// TIA Portal project "DigitalTwin_Selecao_de_Pecas" (V14)
// Trabalho de conclusão de curso, um gêmeo digital de um processo de seleção de peças em uma transportadora

(* hardware
DEVICE "S7-1200 station_3"  S7-1200 Station
   slot 0: "Rack_0"  S7-1200 Rack  Rack  V1.0
   slot 1: "S71200 Físico"  CPU 1214C DC/DC/DC  6ES7 214-1AG40-0XB0  V4.2
   slot 3: "AQ 1x12BIT_1"  AQ1 signal board  6ES7 232-4HA30-0XB0  V1.0
DEVICE "S71500/ET200MP station_2"  S7-1500 station
   slot 0: "Rail_0"  Rack  6ES7 590-1***0-0AA0
   slot 1: "PLCSim Adavanced"  CPU 1511-1 PN  6ES7 511-1AK01-0AB0  V2.1
      slot 3: "CPU display_1"  6ES7591-1AA00-0AA0
*)

// ===== PLC "S71200 Físico"  CPU 1214C DC/DC/DC =====

VAR_GLOBAL   // PLC tag table "Default tag table"
   "System_Byte" AT %MB1 : Byte;
   "FirstScan" AT %M1.0 : Bool;
   "DiagStatusUpdate" AT %M1.1 : Bool;
   "AlwaysTRUE" AT %M1.2 : Bool;
   "AlwaysFALSE" AT %M1.3 : Bool;
   "System_Byte(1)" AT %MB1 : Byte;
   "Clock_Byte" AT %MB0 : Byte;
   "Clock_10Hz" AT %M0.0 : Bool;
   "Clock_5Hz" AT %M0.1 : Bool;
   "Clock_2.5Hz" AT %M0.2 : Bool;
   "Clock_2Hz" AT %M0.3 : Bool;
   "Clock_1.25Hz" AT %M0.4 : Bool;
   "Clock_1Hz" AT %M0.5 : Bool;
   "Clock_0.625Hz" AT %M0.6 : Bool;
   "Clock_0.5Hz" AT %M0.7 : Bool;
END_VAR

VAR_GLOBAL   // PLC tag table "Entradas Digitais"
   "DIn_ATD001_PrsMat01" AT %I0.0 : Bool;   // Esteira transportadora (ET-111) - Presença de material (tamanho maior)
   "DIn_ATD001_PrsMat02" AT %I0.1 : Bool;   // Esteira transportadora (ET-111) - Presença de material (tamanho médio)
   "DIn_ATD001_PrsMat03" AT %I0.2 : Bool;   // Esteira transportadora (ET-111) - Presença de material (tamanho menor)
   "DIn_ATD001_PrsMat04" AT %I0.3 : Bool;   // Esteira transportadora (ET-111) - Presença de material (Capacitivo)
   "DIn_ATD001_PrsMat05" AT %I0.4 : Bool;   // Esteira transportadora (ET-111) - Presença de material (Indutivo)
   "DIn_ATD001_PrsMat06" AT %I0.5 : Bool;   // Esteira transportadora (ET-111) - Presença de material (Setor A)
   "DIn_ATD001_PrsMat07" AT %I0.6 : Bool;   // Esteira transportadora (ET-111) - Presença de material (Setor B)
   "DIn_ATD001_PrsMat08" AT %I0.7 : Bool;   // Esteira transportadora (ET-111) - Presença de material (Setor C)
   "DIn_ATD001_PrsMat09" AT %I1.0 : Bool;   // Esteira transportadora (ET-111) - Presença de material (Setor D)
   "Din_Geral_AtvEmg" AT %I1.1 : Bool;   // Geral - Ativa condição de emergência [NF]
   "Din_Geral_AtvRst" AT %I1.2 : Bool;   // Geral - Ativa reset
END_VAR

VAR_GLOBAL   // PLC tag table "Saídas Analógicas"
   "Dou_ATD001_LigElm" AT %QW64 : UInt;   // Esteira transportadora (ET-111) - Liga elemento (Esteira A)
END_VAR

VAR_GLOBAL   // PLC tag table "Saídas Digitais"
   "Dou_ATD002_AvnElm" AT %Q0.0 : Bool;   // Pistão Separador A (PI-111) - Avança elemento
   "Dou_ATD003_AvnElm" AT %Q0.1 : Bool;   // Pistão Separador B (PI-112) - Avança elemento
   "Dou_ATD004_AvnElm" AT %Q0.2 : Bool;   // Pistão Separador C (PI-113) - Avança elemento
   "Dou_ATD004_RcuElm" AT %Q0.3 : Bool;   // Pistão Separador C (PI-113) - Recua elemento
END_VAR

// folder: System blocks/Program resources

DATA_BLOCK "EES001_DlyDsv01"   // DB4
{ S7_Optimized_Access := 'TRUE' }
AUTHOR : Simatic
FAMILY : IEC
NAME : IEC_TMR
VERSION : 1.0
// stored: InstanceOfName IEC_TIMER
"IEC_TIMER"
BEGIN
END_DATA_BLOCK

// folder: VARIÁVEIS/0 - Gerais

DATA_BLOCK "EDG"   // DB1
TITLE = Detecção de Bordas
{ S7_Optimized_Access := 'TRUE' }
VERSION : 0.1
   VAR
      GRP001_DtcPos01 : Bool;   // Geral - Detecção positiva
      EES001_DtcPos01 : Bool;   // Selecionador de Peças - Detecção positiva
      EES001_DtcPos02 : Bool;   // Selecionador de Peças - Detecção positiva (Aux)
      EES001_DtcPos03 : Bool;   // Selecionador de Peças - Detecção positiva (Tempo de transporte)
   END_VAR
BEGIN
END_DATA_BLOCK

DATA_BLOCK "TMR"   // DB2
TITLE = Temporizadores
{ S7_Optimized_Access := 'TRUE' }
VERSION : 0.1
   VAR
      EES001_DlyAtv01 : IEC_TIMER;   // Selecionador de Peças - Atraso para ativar
      EES001_DlyAtv02 : IEC_TIMER;   // Selecionador de Peças - Atraso para ativar
      EES001_DlyAtv03 : IEC_TIMER;   // Selecionador de Peças - Atraso para ativar
      ATD003_DlyAtv01 : IEC_TIMER;   // Pistão Separador B - Atraso para ativar
      EES001_DlyDsv01 : IEC_TIMER;   // Selecionador de Peças - Atraso para desativar
      EES001_DlyDsv02 : IEC_TIMER;   // Selecionador de Peças - Atraso para desativar (Recuar Pistão C)
      ATD004_DlyAtv01 : IEC_TIMER;   // Pistão Separador C - Atraso para ativar (Avançar)
      EES001_DlyAtv04 : IEC_TIMER;   // Selecionador de Peças - Atraso para ativar (Tempo de transporte)
   END_VAR
BEGIN
END_DATA_BLOCK

DATA_BLOCK "CTR"   // DB3
TITLE = Contadores
{ S7_Optimized_Access := 'TRUE' }
VERSION : 0.1
   VAR
      EES001_CntUnd01 : IEC_UCOUNTER;   // Selecionador de Peças - Conta unidades (Setor A)
      EES001_CntUnd02 : IEC_UCOUNTER;   // Selecionador de Peças - Conta unidades (Setor B)
      EES001_CntUnd03 : IEC_UCOUNTER;   // Selecionador de Peças - Conta unidades (Setor C)
      EES001_CntUnd04 : IEC_UCOUNTER;   // Selecionador de Peças - Conta unidades (Setor D)
   END_VAR
BEGIN
END_DATA_BLOCK

// folder: VARIÁVEIS/1 - Comandos

DATA_BLOCK "CmdEsp"   // DB110
{ S7_Optimized_Access := 'FALSE' }
VERSION : 0.1
BEGIN
END_DATA_BLOCK

DATA_BLOCK "CmdGrp"   // DB120
{ S7_Optimized_Access := 'FALSE' }
VERSION : 0.1
   VAR
      GRP001 : Struct   // Geral
         RrmElm : Bool := false;   // Geral - Rearma Elemento
         SelAut : Bool := false;   // Geral - Seleciona modo automático para todos atuadores
         SelMaa : Bool := false;   // Geral - Seleciona modo manual para todos atuadores
         xd0r3 : Bool := false;   // Reserva
         xd0r4 : Bool := false;   // Reserva
         xd0r5 : Bool := false;   // Reserva
         xd0r6 : Bool := false;   // Reserva
         xd0r7 : Bool := false;   // Reserva
         xd1r0 : Bool := false;   // Reserva
         xd1r1 : Bool := false;   // Reserva
         xd1r2 : Bool := false;   // Reserva
         xd1r3 : Bool := false;   // Reserva
         xd1r4 : Bool := false;   // Reserva
         xd1r5 : Bool := false;   // Reserva
         xd1r6 : Bool := false;   // Reserva
         xd1r7 : Bool := false;   // Reserva
      END_STRUCT;
   END_VAR
BEGIN
END_DATA_BLOCK

DATA_BLOCK "CmdAtd"   // DB130
TITLE = Comandos
{ S7_Optimized_Access := 'FALSE' }
VERSION : 0.1
   VAR
      ATD001 : Struct   // Esteira Transportadora (ET-111)
         SelAut : Bool;   // Esteira Transportadora (ET-111) - Seleciona modo automático
         SelMaa : Bool := false;   // Esteira Transportadora (ET-111) - Seleciona modo manual
         LigElm : Bool := false;   // Esteira Transportadora (ET-111) - Liga elemento
         DsgElm : Bool := false;   // Esteira Transportadora (ET-111) - Desliga elemento
         xd0r4 : Bool := false;   // Reserva
         xd0r5 : Bool := false;   // Reserva
         xd0r6 : Bool := false;   // Reserva
         xd0r7 : Bool := false;   // Reserva
         xd1r0 : Bool;   // Reserva
         xd1r1 : Bool := false;   // Reserva
         xd1r2 : Bool := false;   // Reserva
         xd1r3 : Bool := false;   // Reserva
         xd1r4 : Bool := false;   // Reserva
         xd1r5 : Bool := false;   // Reserva
         xd1r6 : Bool := false;   // Reserva
         xd1r7 : Bool := false;   // Reserva
      END_STRUCT;
      ATD002 : Struct   // Pistão Separador A (PI-111)
         SelAut : Bool := false;   // Pistão Separador A (PI-111) - Seleciona modo automático
         SelMaa : Bool := false;   // Pistão Separador A (PI-111) - Seleciona modo manual
         AvnElm : Bool := false;   // Pistão Separador A (PI-111) - Avança elemento
         RcuElm : Bool := false;   // Pistão Separador A (PI-111) - Recua elemento
         xd0r4 : Bool := false;   // Reserva
         xd0r5 : Bool := false;   // Reserva
         xd0r6 : Bool := false;   // Reserva
         xd0r7 : Bool := false;   // Reserva
         xd1r0 : Bool := false;   // Reserva
         xd1r1 : Bool := false;   // Reserva
         xd1r2 : Bool := false;   // Reserva
         xd1r3 : Bool := false;   // Reserva
         xd1r4 : Bool := false;   // Reserva
         xd1r5 : Bool := false;   // Reserva
         xd1r6 : Bool := false;   // Reserva
         xd1r7 : Bool := false;   // Reserva
      END_STRUCT;
      ATD003 : Struct   // Pistão Separador B (PI-112)
         SelAut : Bool := false;   // Pistão Separador B (PI-112) - Seleciona modo automático
         SelMaa : Bool := false;   // Pistão Separador B (PI-112) - Seleciona modo manual
         AvnElm : Bool := false;   // Pistão Separador B (PI-112) - Avança elemento
         RcuElm : Bool := false;   // Pistão Separador B (PI-112) - Recua elemento
         xd0r4 : Bool := false;   // Reserva
         xd0r5 : Bool := false;   // Reserva
         xd0r6 : Bool := false;   // Reserva
         xd0r7 : Bool := false;   // Reserva
         xd1r0 : Bool := false;   // Reserva
         xd1r1 : Bool := false;   // Reserva
         xd1r2 : Bool := false;   // Reserva
         xd1r3 : Bool := false;   // Reserva
         xd1r4 : Bool := false;   // Reserva
         xd1r5 : Bool := false;   // Reserva
         xd1r6 : Bool := false;   // Reserva
         xd1r7 : Bool := false;   // Reserva
      END_STRUCT;
      ATD004 : Struct   // Pistão Separador C (PI-113)
         SelAut : Bool := false;   // Pistão Separador C (PI-113) - Seleciona modo automático
         SelMaa : Bool := false;   // Pistão Separador C (PI-113) - Seleciona modo manual
         AvnElm : Bool := false;   // Pistão Separador C (PI-113) - Avança elemento
         RcuElm : Bool := false;   // Pistão Separador C (PI-113) - Recua elemento
         xd0r4 : Bool := false;   // Reserva
         xd0r5 : Bool := false;   // Reserva
         xd0r6 : Bool := false;   // Reserva
         xd0r7 : Bool := false;   // Reserva
         xd1r0 : Bool := false;   // Reserva
         xd1r1 : Bool := false;   // Reserva
         xd1r2 : Bool := false;   // Reserva
         xd1r3 : Bool := false;   // Reserva
         xd1r4 : Bool := false;   // Reserva
         xd1r5 : Bool := false;   // Reserva
         xd1r6 : Bool := false;   // Reserva
         xd1r7 : Bool := false;   // Reserva
      END_STRUCT;
   END_VAR
BEGIN
END_DATA_BLOCK

DATA_BLOCK "CmdEes"   // DB160
{ S7_Optimized_Access := 'FALSE' }
VERSION : 0.1
   VAR
      EES001 : Struct   // Selecionador de Peças
         RrmElm : Bool := false;   // Selecionador de Peças - Rearma Elmento
         RmvPcs01 : Bool := false;   // Selecionador de Peças - Remove Peças (Setor A)
         RmvPcs02 : Bool := false;   // Selecionador de Peças - Remove Peças (Setor B)
         RmvPcs03 : Bool := false;   // Selecionador de Peças - Remove Peças (Setor C)
         RmvPcs04 : Bool := false;   // Selecionador de Peças - Remove Peças (Setor D)
         RstPcs : Bool := false;   // Selecionador de Peças - Reseta quantidade de Peças
         xd0r6 : Bool := false;   // Reserva
         xd0r7 : Bool := false;   // Reserva
         xd1r0 : Bool := false;   // Reserva
         xd1r1 : Bool := false;   // Reserva
         xd1r2 : Bool := false;   // Reserva
         xd1r3 : Bool := false;   // Reserva
         xd1r4 : Bool := false;   // Reserva
         xd1r5 : Bool := false;   // Reserva
         xd1r6 : Bool := false;   // Reserva
         xd1r7 : Bool := false;   // Reserva
      END_STRUCT;
   END_VAR
BEGIN
END_DATA_BLOCK

// folder: VARIÁVEIS/2 - Estados

DATA_BLOCK "SttEsp"   // DB210
{ S7_Optimized_Access := 'FALSE' }
VERSION : 0.1
BEGIN
END_DATA_BLOCK

DATA_BLOCK "SttGrp"   // DB220
{ S7_Optimized_Access := 'FALSE' }
VERSION : 0.1
   VAR
      GRP001 : Struct   // Geral
         xd0r0 : Bool := false;   // Reserva
         xd0r1 : Bool := false;   // Reserva
         xd0r2 : Bool := false;   // Reserva
         xd0r3 : Bool := false;   // Reserva
         xd0r4 : Bool := false;   // Reserva
         xd0r5 : Bool := false;   // Reserva
         xd0r6 : Bool := false;   // Reserva
         xd0r7 : Bool := false;   // Reserva
         xd1r0 : Bool := false;   // Reserva
         xd1r1 : Bool := false;   // Reserva
         xd1r2 : Bool := false;   // Reserva
         xd1r3 : Bool := false;   // Reserva
         xd1r4 : Bool := false;   // Reserva
         xd1r5 : Bool := false;   // Reserva
         xd1r6 : Bool := false;   // Reserva
         xd1r7 : Bool := false;   // Reserva
      END_STRUCT;
   END_VAR
BEGIN
END_DATA_BLOCK

DATA_BLOCK "SttAtd"   // DB230
TITLE = Estados de Atuadores
{ S7_Optimized_Access := 'FALSE' }
VERSION : 0.1
   VAR
      ATD001 : Struct   // Esteira Transportadora (ET-111)
         AutSel : Bool := false;   // Esteira Transportadora (ET-111) - Modo automático selecionado
         MaaSel : Bool := false;   // Esteira Transportadora (ET-111) - Modo manual selecionado
         ElmLig : Bool := false;   // Esteira Transportadora (ET-111) - Elemento ligado
         BlqLig : Bool := false;   // Esteira Transportadora (ET-111) - Bloqueado para ligar
         xd0r4 : Bool := false;   // Reserva
         xd0r5 : Bool := false;   // Reserva
         xd0r6 : Bool := false;   // Reserva
         xd0r7 : Bool := false;   // Reserva
         xd1r0 : Bool := false;   // Reserva
         xd1r1 : Bool := false;   // Reserva
         xd1r2 : Bool := false;   // Reserva
         xd1r3 : Bool := false;   // Reserva
         xd1r4 : Bool := false;   // Reserva
         xd1r5 : Bool := false;   // Reserva
         xd1r6 : Bool := false;   // Reserva
         xd1r7 : Bool := false;   // Reserva
      END_STRUCT;
      ATD002 : Struct   // Pistão Separador A (PI-111)
         AutSel : Bool := false;   // Pistão Separador A (PI-111) - Modo automático selecionado
         MaaSel : Bool := false;   // Pistão Separador A (PI-111) - Modo manual selecionado
         PosAvn : Bool := false;   // Pistão Separador A (PI-111) - Elemento avançado
         BlqAvn : Bool := false;   // Pistão Separador A (PI-111) - Bloqueado para avançar
         xd0r4 : Bool := false;   // Reserva
         xd0r5 : Bool := false;   // Reserva
         xd0r6 : Bool := false;   // Reserva
         xd0r7 : Bool := false;   // Reserva
         xd1r0 : Bool := false;   // Reserva
         xd1r1 : Bool := false;   // Reserva
         xd1r2 : Bool := false;   // Reserva
         xd1r3 : Bool := false;   // Reserva
         xd1r4 : Bool := false;   // Reserva
         xd1r5 : Bool := false;   // Reserva
         xd1r6 : Bool := false;   // Reserva
         xd1r7 : Bool := false;   // Reserva
      END_STRUCT;
      ATD003 : Struct   // Pistão Separador B (PI-112)
         AutSel : Bool := false;   // Pistão Separador B (PI-112) - Modo automático selecionado
         MaaSel : Bool := false;   // Pistão Separador B (PI-112) - Modo manual selecionado
         PosAvn : Bool := false;   // Pistão Separador B (PI-112) - Elemento avançado
         BlqAvn : Bool := false;   // Pistão Separador B (PI-112) - Bloqueado para Bloqueado para avançar
         xd0r4 : Bool := false;   // Reserva
         xd0r5 : Bool := false;   // Reserva
         xd0r6 : Bool := false;   // Reserva
         xd0r7 : Bool := false;   // Reserva
         xd1r0 : Bool := false;   // Reserva
         xd1r1 : Bool := false;   // Reserva
         xd1r2 : Bool := false;   // Reserva
         xd1r3 : Bool := false;   // Reserva
         xd1r4 : Bool := false;   // Reserva
         xd1r5 : Bool := false;   // Reserva
         xd1r6 : Bool := false;   // Reserva
         xd1r7 : Bool := false;   // Reserva
      END_STRUCT;
      ATD004 : Struct   // Pistão Separador C (PI-113)
         AutSel : Bool := false;   // Pistão Separador C (PI-113) - Modo automático selecionado
         MaaSel : Bool := false;   // Pistão Separador C (PI-113) - Modo manual selecionado
         PosAvn : Bool := false;   // Pistão Separador C (PI-113) - Elemento avançado
         BlqAvn : Bool := false;   // Pistão Separador C (PI-113) - Bloqueado para avançar
         PosRcu : Bool := false;   // Pistão Separador C (PI-113) - Elemento recuado
         BlqRcu : Bool := false;   // Pistão Separador C (PI-113) - Bloqueado para recuar
         xd0r6 : Bool := false;   // Reserva
         xd0r7 : Bool := false;   // Reserva
         xd1r0 : Bool := false;   // Reserva
         xd1r1 : Bool := false;   // Reserva
         xd1r2 : Bool := false;   // Reserva
         xd1r3 : Bool := false;   // Reserva
         xd1r4 : Bool := false;   // Reserva
         xd1r5 : Bool := false;   // Reserva
         xd1r6 : Bool := false;   // Reserva
         xd1r7 : Bool := false;   // Reserva
      END_STRUCT;
   END_VAR
BEGIN
END_DATA_BLOCK

DATA_BLOCK "SttEes"   // DB260
{ S7_Optimized_Access := 'FALSE' }
VERSION : 0.1
   VAR
      EES001 : Struct   // Selecionador de Peças
         ElmDef : Bool := false;   // Selecionador de Peças - Elmento com Defeito
         xd0r1 : Bool := false;   // Reserva
         xd0r2 : Bool := false;   // Reserva
         xd0r3 : Bool := false;   // Reserva
         xd0r4 : Bool := false;   // Reserva
         xd0r5 : Bool := false;   // Reserva
         xd0r6 : Bool := false;   // Reserva
         xd0r7 : Bool := false;   // Reserva
         xd1r0 : Bool := false;   // Reserva
         xd1r1 : Bool := false;   // Reserva
         xd1r2 : Bool := false;   // Reserva
         xd1r3 : Bool := false;   // Reserva
         xd1r4 : Bool := false;   // Reserva
         xd1r5 : Bool := false;   // Reserva
         xd1r6 : Bool := false;   // Reserva
         xd1r7 : Bool := false;   // Reserva
      END_STRUCT;
   END_VAR
BEGIN
END_DATA_BLOCK

// folder: VARIÁVEIS/3 - Alarmes

DATA_BLOCK "AlrEsp"   // DB310
{ S7_Optimized_Access := 'FALSE' }
VERSION : 0.1
BEGIN
END_DATA_BLOCK

DATA_BLOCK "AlrGrp"   // DB320
{ S7_Optimized_Access := 'FALSE' }
VERSION : 0.1
   VAR
      GRP001 : Struct   // Geral
         EmgAtv : Bool := false;   // Geral - Condição de Emergência Ativada
         xd0r1 : Bool := false;   // Reserva
         xd0r2 : Bool := false;   // Reserva
         xd0r3 : Bool := false;   // Reserva
         xd0r4 : Bool := false;   // Reserva
         xd0r5 : Bool := false;   // Reserva
         xd0r6 : Bool := false;   // Reserva
         xd0r7 : Bool := false;   // Reserva
         xd1r0 : Bool := false;   // Reserva
         xd1r1 : Bool := false;   // Reserva
         xd1r2 : Bool := false;   // Reserva
         xd1r3 : Bool := false;   // Reserva
         xd1r4 : Bool := false;   // Reserva
         xd1r5 : Bool := false;   // Reserva
         xd1r6 : Bool := false;   // Reserva
         xd1r7 : Bool := false;   // Reserva
      END_STRUCT;
   END_VAR
BEGIN
END_DATA_BLOCK

DATA_BLOCK "AlrAtd"   // DB330
TITLE = Alarmes de Atuadores
{ S7_Optimized_Access := 'FALSE' }
VERSION : 0.1
   VAR
      ATD001 : Struct   // Esteira Transportadora (ET-111)
         xd0r0 : Bool := false;   // Reserva
         xd0r1 : Bool := false;   // Reserva
         xd0r2 : Bool := false;   // Reserva
         xd0r3 : Bool := false;   // Reserva
         xd0r4 : Bool := false;   // Reserva
         xd0r5 : Bool := false;   // Reserva
         xd0r6 : Bool := false;   // Reserva
         xd0r7 : Bool := false;   // Reserva
         xd1r0 : Bool := false;   // Reserva
         xd1r1 : Bool := false;   // Reserva
         xd1r2 : Bool := false;   // Reserva
         xd1r3 : Bool := false;   // Reserva
         xd1r4 : Bool := false;   // Reserva
         xd1r5 : Bool := false;   // Reserva
         xd1r6 : Bool := false;   // Reserva
         xd1r7 : Bool := false;   // Reserva
      END_STRUCT;
      ATD002 : Struct   // Pistão Separador A (PI-111)
         xd0r0 : Bool := false;   // Reserva
         xd0r1 : Bool := false;   // Reserva
         xd0r2 : Bool := false;   // Reserva
         xd0r3 : Bool := false;   // Reserva
         xd0r4 : Bool := false;   // Reserva
         xd0r5 : Bool := false;   // Reserva
         xd0r6 : Bool := false;   // Reserva
         xd0r7 : Bool := false;   // Reserva
         xd1r0 : Bool := false;   // Reserva
         xd1r1 : Bool := false;   // Reserva
         xd1r2 : Bool := false;   // Reserva
         xd1r3 : Bool := false;   // Reserva
         xd1r4 : Bool := false;   // Reserva
         xd1r5 : Bool := false;   // Reserva
         xd1r6 : Bool := false;   // Reserva
         xd1r7 : Bool := false;   // Reserva
      END_STRUCT;
      ATD003 : Struct   // Pistão Separador B (PI-112)
         xd0r0 : Bool := false;   // Reserva
         xd0r1 : Bool := false;   // Reserva
         xd0r2 : Bool := false;   // Reserva
         xd0r3 : Bool := false;   // Reserva
         xd0r4 : Bool := false;   // Reserva
         xd0r5 : Bool := false;   // Reserva
         xd0r6 : Bool := false;   // Reserva
         xd0r7 : Bool := false;   // Reserva
         xd1r0 : Bool := false;   // Reserva
         xd1r1 : Bool := false;   // Reserva
         xd1r2 : Bool := false;   // Reserva
         xd1r3 : Bool := false;   // Reserva
         xd1r4 : Bool := false;   // Reserva
         xd1r5 : Bool := false;   // Reserva
         xd1r6 : Bool := false;   // Reserva
         xd1r7 : Bool := false;   // Reserva
      END_STRUCT;
      ATD004 : Struct   // Pistão Separador C (PI-113)
         xd0r0 : Bool := false;   // Reserva
         xd0r1 : Bool := false;   // Reserva
         xd0r2 : Bool := false;   // Reserva
         xd0r3 : Bool := false;   // Reserva
         xd0r4 : Bool := false;   // Reserva
         xd0r5 : Bool := false;   // Reserva
         xd0r6 : Bool := false;   // Reserva
         xd0r7 : Bool := false;   // Reserva
         xd1r0 : Bool := false;   // Reserva
         xd1r1 : Bool := false;   // Reserva
         xd1r2 : Bool := false;   // Reserva
         xd1r3 : Bool := false;   // Reserva
         xd1r4 : Bool := false;   // Reserva
         xd1r5 : Bool := false;   // Reserva
         xd1r6 : Bool := false;   // Reserva
         xd1r7 : Bool := false;   // Reserva
      END_STRUCT;
   END_VAR
BEGIN
END_DATA_BLOCK

DATA_BLOCK "AlrEes"   // DB360
{ S7_Optimized_Access := 'FALSE' }
VERSION : 0.1
   VAR
      EES001 : Struct   // Selecionador de Peças
         LimExc : Bool := false;   // Selecionador de Peças - Limite Excedido (Mais de uma peça em transporte)
         xd0r1 : Bool := false;   // Reserva
         xd0r2 : Bool := false;   // Reserva
         xd0r3 : Bool := false;   // Reserva
         xd0r4 : Bool := false;   // Reserva
         xd0r5 : Bool := false;   // Reserva
         xd0r6 : Bool := false;   // Reserva
         xd0r7 : Bool := false;   // Reserva
         xd1r0 : Bool := false;   // Reserva
         xd1r1 : Bool := false;   // Reserva
         xd1r2 : Bool := false;   // Reserva
         xd1r3 : Bool := false;   // Reserva
         xd1r4 : Bool := false;   // Reserva
         xd1r5 : Bool := false;   // Reserva
         xd1r6 : Bool := false;   // Reserva
         xd1r7 : Bool := false;   // Reserva
      END_STRUCT;
   END_VAR
BEGIN
END_DATA_BLOCK

// folder: VARIÁVEIS/4 - Intertravamentos

DATA_BLOCK "IlkEsp"   // DB410
{ S7_Optimized_Access := 'FALSE' }
VERSION : 0.1
BEGIN
END_DATA_BLOCK

DATA_BLOCK "IlkGrp"   // DB420
{ S7_Optimized_Access := 'FALSE' }
VERSION : 0.1
   VAR
      GRP001 : Struct   // Geral
         xd0r0 : Bool := false;   // Reserva
         xd0r1 : Bool := false;   // Reserva
         xd0r2 : Bool := false;   // Reserva
         xd0r3 : Bool := false;   // Reserva
         xd0r4 : Bool := false;   // Reserva
         xd0r5 : Bool := false;   // Reserva
         xd0r6 : Bool := false;   // Reserva
         xd0r7 : Bool := false;   // Reserva
         xd1r0 : Bool := false;   // Reserva
         xd1r1 : Bool := false;   // Reserva
         xd1r2 : Bool := false;   // Reserva
         xd1r3 : Bool := false;   // Reserva
         xd1r4 : Bool := false;   // Reserva
         xd1r5 : Bool := false;   // Reserva
         xd1r6 : Bool := false;   // Reserva
         xd1r7 : Bool := false;   // Reserva
      END_STRUCT;
   END_VAR
BEGIN
END_DATA_BLOCK

DATA_BLOCK "IlkAtd"   // DB430
TITLE = Intertravamentos de Atuadores
{ S7_Optimized_Access := 'FALSE' }
VERSION : 0.1
   VAR
      ATD001 : Struct   // Esteira Transportadora (ET-111)
         BlqLig01 : Bool := false;   // Esteira Transportadora (ET-111) - Bloqueado para ligar (Condição de emergência ativada)
         BlqLig02 : Bool := false;   // Esteira Transportadora (ET-111) - Bloqueado para ligar (Todos os Setores Cheios)
         BlqLig03 : Bool := false;   // Esteira Transportadora (ET-111) - Bloqueado para ligar (Selecionador de Peça com defeito)
         xd0r3 : Bool := false;   // Reserva
         xd0r4 : Bool := false;   // Reserva
         xd0r5 : Bool := false;   // Reserva
         xd0r6 : Bool := false;   // Reserva
         xd0r7 : Bool := false;   // Reserva
         xd1r0 : Bool := false;   // Reserva
         xd1r1 : Bool := false;   // Reserva
         xd1r2 : Bool := false;   // Reserva
         xd1r3 : Bool := false;   // Reserva
         xd1r4 : Bool := false;   // Reserva
         xd1r5 : Bool := false;   // Reserva
         xd1r6 : Bool := false;   // Reserva
         xd1r7 : Bool := false;   // Reserva
      END_STRUCT;
      ATD002 : Struct   // Pistão Separador A (PI-111)
         BlqAvn01 : Bool := false;   // Pistão Separador A (PI-111) - Bloqueado para avançar (Condição de emergência ativada)
         BlqAvn02 : Bool := false;   // Pistão Separador A (PI-111) - Bloqueado para avançar (Setor A Cheio)
         BlqAvn03 : Bool := false;   // Reserva
         xd0r3 : Bool := false;   // Reserva
         xd0r4 : Bool := false;   // Reserva
         xd0r5 : Bool := false;   // Reserva
         xd0r6 : Bool := false;   // Reserva
         xd0r7 : Bool := false;   // Reserva
         xd1r0 : Bool := false;   // Reserva
         xd1r1 : Bool := false;   // Reserva
         xd1r2 : Bool := false;   // Reserva
         xd1r3 : Bool := false;   // Reserva
         xd1r4 : Bool := false;   // Reserva
         xd1r5 : Bool := false;   // Reserva
         xd1r6 : Bool := false;   // Reserva
         xd1r7 : Bool := false;   // Reserva
      END_STRUCT;
      ATD003 : Struct   // Pistão Separador B (PI-112)
         BlqAvn01 : Bool := false;   // Pistão Separador B (PI-112) - Bloqueado para avançar (Condição de emergência ativada)
         BlqAvn02 : Bool := false;   // Pistão Separador B (PI-112) - Bloqueado para avançar (Setor B Cheio)
         BlqAvn03 : Bool := false;   // Pistão Separador B (PI-112) - Bloqueado para avançar (Selecionador de Peça com defeito)
         BlqAvn04 : Bool := false;   // Pistão Separador B (PI-112) - Bloqueado para avançar (Pistão Separador A ou B Avançados)
         xd0r4 : Bool := false;   // Reserva
         xd0r5 : Bool := false;   // Reserva
         xd0r6 : Bool := false;   // Reserva
         xd0r7 : Bool := false;   // Reserva
         xd1r0 : Bool := false;   // Reserva
         xd1r1 : Bool := false;   // Reserva
         xd1r2 : Bool := false;   // Reserva
         xd1r3 : Bool := false;   // Reserva
         xd1r4 : Bool := false;   // Reserva
         xd1r5 : Bool := false;   // Reserva
         xd1r6 : Bool := false;   // Reserva
         xd1r7 : Bool := false;   // Reserva
      END_STRUCT;
      ATD004 : Struct   // Pistão Separador C (PI-113)
         BlqAvn01 : Bool := false;   // Pistão Separador C (PI-113) - Bloqueado para avançar (Condição de emergência ativada)
         BlqAvn02 : Bool := false;   // Pistão Separador C (PI-113) - Bloqueado para avançar (Setor C Cheio)
         BlqAvn03 : Bool := false;   // Pistão Separador C (PI-113) - Bloqueado para avançar (Selecionador de Peça com defeito)
         BlqAvn04 : Bool := false;   // Pistão Separador C (PI-113) - Bloqueado para avançar (Pistão Separador B Avançado)
         xd0r4 : Bool := false;   // Reserva
         xd0r5 : Bool := false;   // Reserva
         xd0r6 : Bool := false;   // Reserva
         xd0r7 : Bool := false;   // Reserva
         xd1r0 : Bool := false;   // Reserva
         xd1r1 : Bool := false;   // Reserva
         xd1r2 : Bool := false;   // Reserva
         xd1r3 : Bool := false;   // Reserva
         xd1r4 : Bool := false;   // Reserva
         xd1r5 : Bool := false;   // Reserva
         xd1r6 : Bool := false;   // Reserva
         xd1r7 : Bool := false;   // Reserva
      END_STRUCT;
   END_VAR
BEGIN
END_DATA_BLOCK

DATA_BLOCK "IlkEes"   // DB460
{ S7_Optimized_Access := 'FALSE' }
VERSION : 0.1
BEGIN
END_DATA_BLOCK

// folder: VARIÁVEIS/5 - Auxiliar Digital

DATA_BLOCK "DAuEsp"   // DB510
{ S7_Optimized_Access := 'FALSE' }
VERSION : 0.1
   VAR
      ESP001 : Struct   // CPU do CLP
         Pls1seg : Bool := false;   // CPU do CLP - Pulso de 1 segundo
         xd0r1 : Bool := false;   // Reserva
         xd0r2 : Bool := false;   // Reserva
         xd0r3 : Bool := false;   // Reserva
         xd0r4 : Bool := false;   // Reserva
         xd0r5 : Bool := false;   // Reserva
         xd0r6 : Bool := false;   // Reserva
         xd0r7 : Bool := false;   // Reserva
         xd1r0 : Bool := false;   // Reserva
         xd1r1 : Bool := false;   // Reserva
         xd1r2 : Bool := false;   // Reserva
         xd1r3 : Bool := false;   // Reserva
         xd1r4 : Bool := false;   // Reserva
         xd1r5 : Bool := false;   // Reserva
         xd1r6 : Bool := false;   // Reserva
         xd1r7 : Bool := false;   // Reserva
      END_STRUCT;
   END_VAR
BEGIN
END_DATA_BLOCK

DATA_BLOCK "DAuGrp"   // DB520
{ S7_Optimized_Access := 'FALSE' }
VERSION : 0.1
BEGIN
END_DATA_BLOCK

DATA_BLOCK "DAuAtd"   // DB530
TITLE = Auxiliares digitais de atuadores
{ S7_Optimized_Access := 'FALSE' }
VERSION : 0.1
   VAR
      ATD001 : Struct   // Esteira Transportadora (ET-111)
         AutLig : Bool := false;   // Esteira Transportadora (ET-111) - Liga via modo automático
         MaaLig : Bool := false;   // Esteira Transportadora (ET-111) - Liga via modo manual
         xd0r2 : Bool := false;   // Reserva
         xd0r3 : Bool := false;   // Reserva
         xd0r4 : Bool := false;   // Reserva
         xd0r5 : Bool := false;   // Reserva
         xd0r6 : Bool := false;   // Reserva
         xd0r7 : Bool := false;   // Reserva
         xd1r0 : Bool := false;   // Reserva
         xd1r1 : Bool := false;   // Reserva
         xd1r2 : Bool := false;   // Reserva
         xd1r3 : Bool := false;   // Reserva
         xd1r4 : Bool := false;   // Reserva
         xd1r5 : Bool := false;   // Reserva
         xd1r6 : Bool := false;   // Reserva
         xd1r7 : Bool := false;   // Reserva
      END_STRUCT;
      ATD002 : Struct   // Pistão Separador A (PI-111)
         AutAvn : Bool := false;   // Pistão Separador A (PI-111) - Avança via modo automático
         MaaAvn : Bool := false;   // Pistão Separador A (PI-111) - Avança via modo manual
         xd0r2 : Bool := false;   // Reserva
         xd0r3 : Bool := false;   // Reserva
         xd0r4 : Bool := false;   // Reserva
         xd0r5 : Bool := false;   // Reserva
         xd0r6 : Bool := false;   // Reserva
         xd0r7 : Bool := false;   // Reserva
         xd1r0 : Bool := false;   // Reserva
         xd1r1 : Bool := false;   // Reserva
         xd1r2 : Bool := false;   // Reserva
         xd1r3 : Bool := false;   // Reserva
         xd1r4 : Bool := false;   // Reserva
         xd1r5 : Bool := false;   // Reserva
         xd1r6 : Bool := false;   // Reserva
         xd1r7 : Bool := false;   // Reserva
      END_STRUCT;
      ATD003 : Struct   // Pistão Separador B (PI-112)
         AutAvn : Bool := false;   // Pistão Separador B (PI-112) - Avança via modo automático
         MaaAvn : Bool := false;   // Pistão Separador B (PI-112) - Avança via modo manual
         xd0r2 : Bool := false;   // Reserva
         xd0r3 : Bool := false;   // Reserva
         xd0r4 : Bool := false;   // Reserva
         xd0r5 : Bool := false;   // Reserva
         xd0r6 : Bool := false;   // Reserva
         xd0r7 : Bool := false;   // Reserva
         xd1r0 : Bool := false;   // Reserva
         xd1r1 : Bool := false;   // Reserva
         xd1r2 : Bool := false;   // Reserva
         xd1r3 : Bool := false;   // Reserva
         xd1r4 : Bool := false;   // Reserva
         xd1r5 : Bool := false;   // Reserva
         xd1r6 : Bool := false;   // Reserva
         xd1r7 : Bool := false;   // Reserva
      END_STRUCT;
      ATD004 : Struct   // Pistão Separador C (PI-113)
         AutAvn : Bool := false;   // Pistão Separador C (PI-113) - Avança via modo automático
         MaaAvn : Bool := false;   // Pistão Separador C (PI-113) - Avança via modo manual
         AutRcu : Bool := false;   // Pistão Separador C (PI-113) - Recua via modo automático
         MaaRcu : Bool := false;   // Pistão Separador C (PI-113) - Recua via modo manual
         xd0r4 : Bool := false;   // Reserva
         xd0r5 : Bool := false;   // Reserva
         xd0r6 : Bool := false;   // Reserva
         xd0r7 : Bool := false;   // Reserva
         xd1r0 : Bool := false;   // Reserva
         xd1r1 : Bool := false;   // Reserva
         xd1r2 : Bool := false;   // Reserva
         xd1r3 : Bool := false;   // Reserva
         xd1r4 : Bool := false;   // Reserva
         xd1r5 : Bool := false;   // Reserva
         xd1r6 : Bool := false;   // Reserva
         xd1r7 : Bool := false;   // Reserva
      END_STRUCT;
   END_VAR
BEGIN
END_DATA_BLOCK

DATA_BLOCK "DauEes"   // DB560
{ S7_Optimized_Access := 'FALSE' }
VERSION : 0.1
   VAR
      EES001_Sel : Struct   // Selecionador de Peças - Peças selecionadas para cada setor
         SetAPec01 : Bool;   // Selecionador de Peças - Setor A aceita Metal Pequeno
         SetAPec02 : Bool := false;   // Selecionador de Peças - Setor A aceita Metal Médio
         SetAPec03 : Bool := false;   // Selecionador de Peças - Setor A aceita Metal Grande
         SetAPec04 : Bool := false;   // Selecionador de Peças - Setor A aceita Plástico Pequeno
         SetAPec05 : Bool := false;   // Selecionador de Peças - Setor A aceita Plástico Médio
         SetAPec06 : Bool := false;   // Selecionador de Peças - Setor A aceita Plástico Grande
         SetBPec01 : Bool;   // Selecionador de Peças - Setor B aceita Metal Pequeno
         SetBPec02 : Bool;   // Selecionador de Peças - Setor B aceita Metal Médio
         SetBPec03 : Bool;   // Selecionador de Peças - Setor B aceita Metal Grande
         SetBPec04 : Bool;   // Selecionador de Peças - Setor B aceita Plástico Pequeno
         SetBPec05 : Bool;   // Selecionador de Peças - Setor B aceita Plástico Médio
         SetBPec06 : Bool;   // Selecionador de Peças - Setor B aceita Plástico Grande
         SetCPec01 : Bool;   // Selecionador de Peças - Setor C aceita Metal Pequeno
         SetCPec02 : Bool;   // Selecionador de Peças - Setor C aceita Metal Médio
         SetCPec03 : Bool;   // Selecionador de Peças - Setor C aceita Metal Grande
         SetCPec04 : Bool;   // Selecionador de Peças - Setor C aceita Plástico Pequeno
         SetCPec05 : Bool;   // Selecionador de Peças - Setor C aceita Plástico Médio
         SetCPec06 : Bool;   // Selecionador de Peças - Setor C aceita Plástico Grande
         SetDPec01 : Bool;   // Selecionador de Peças - Setor D aceita Metal Pequeno
         SetDPec02 : Bool;   // Selecionador de Peças - Setor D aceita Metal Médio
         SetDPec03 : Bool;   // Selecionador de Peças - Setor D aceita Metal Grande
         SetDPec04 : Bool;   // Selecionador de Peças - Setor D aceita Plástico Pequeno
         SetDPec05 : Bool;   // Selecionador de Peças - Setor D aceita Plástico Médio
         SetDPec06 : Bool;   // Selecionador de Peças - Setor D aceita Plástico Grande
      END_STRUCT;
      EES001_NewPec : Bool;   // Selecionador de Peças - Nova Peça em transporte
      EES001 : Struct   // Selecionador de Peças
         LigEst : Bool := false;   // Selecionador de Peças - Liga Esteira
         AvnPiA : Bool := false;   // Selecionador de Peças - Avança Pistão Separador A
         AvnPiB : Bool := false;   // Selecionador de Peças - Avança Pistão Separador B
         AvnPiC : Bool := false;   // Selecionador de Peças - Avança Pistão Separador C
         RcuPiC : Bool := false;   // Selecionador de Peças - Recua Pistão Separador C
         xd0r5 : Bool := false;   // Reserva
         xd0r6 : Bool := false;   // Reserva
         xd0r7 : Bool := false;   // Reserva
         xd1r0 : Bool := false;   // Reserva
         xd1r1 : Bool := false;   // Reserva
         xd1r2 : Bool := false;   // Reserva
         xd1r3 : Bool := false;   // Reserva
         xd1r4 : Bool := false;   // Reserva
         xd1r5 : Bool := false;   // Reserva
         xd1r6 : Bool := false;   // Reserva
         xd1r7 : Bool := false;   // Reserva
      END_STRUCT;
   END_VAR
BEGIN
END_DATA_BLOCK

// folder: VARIÁVEIS/6 - Auxiliar Analógica

DATA_BLOCK "AAuEsp"   // DB610
{ S7_Optimized_Access := 'FALSE' }
VERSION : 0.1
   VAR
      ESP001_DmxFrm : DWord;   // CPU do CLP - Frame a ser demultiplexado
      ESP001_SinAtv : Real;   // CPU do CLP - Sinal de atividade do CLP
   END_VAR
BEGIN
END_DATA_BLOCK

DATA_BLOCK "AAuGrp"   // DB620
{ S7_Optimized_Access := 'FALSE' }
VERSION : 0.1
BEGIN
END_DATA_BLOCK

DATA_BLOCK "AAuAtd"   // DB630
TITLE = Auxiliares Analógicas de Atuadores
{ S7_Optimized_Access := 'FALSE' }
VERSION : 0.1
BEGIN
END_DATA_BLOCK

DATA_BLOCK "AAuEes"   // DB660
{ S7_Optimized_Access := 'FALSE' }
VERSION : 0.1
   VAR
      EES001_TmpTrp : Time;   // Selecionador de Peças - Tempo de Transporte
   END_VAR
BEGIN
END_DATA_BLOCK

// folder: VARIÁVEIS/7 - Grandezas Analógicas

DATA_BLOCK "AnaEsp"   // DB710
{ S7_Optimized_Access := 'FALSE' }
VERSION : 0.1
BEGIN
END_DATA_BLOCK

DATA_BLOCK "AnaGrp"   // DB720
{ S7_Optimized_Access := 'FALSE' }
VERSION : 0.1
BEGIN
END_DATA_BLOCK

DATA_BLOCK "AnaAtd"   // DB730
TITLE = Grandezas Analógicas de Atuadores
{ S7_Optimized_Access := 'FALSE' }
VERSION : 0.1
BEGIN
END_DATA_BLOCK

DATA_BLOCK "AnaEes"   // DB760
{ S7_Optimized_Access := 'FALSE' }
VERSION : 0.1
   VAR
      EES001_QtdPec01 : UInt;   // Selecionador de Peças - Quantidade de Peças (Setor A)
      EES001_QtdPec02 : UInt := 0;   // Selecionador de Peças - Quantidade de Peças (Setor B)
      EES001_QtdPec03 : UInt := 0;   // Selecionador de Peças - Quantidade de Peças (Setor C)
      EES001_QtdPec04 : UInt := 0;   // Selecionador de Peças - Quantidade de Peças (Setor D)
   END_VAR
BEGIN
END_DATA_BLOCK

// folder: VARIÁVEIS/8 - Parâmetros

DATA_BLOCK "ParEsp"   // DB810
{ S7_Optimized_Access := 'FALSE' }
VERSION : 0.1
BEGIN
END_DATA_BLOCK

DATA_BLOCK "ParGrp"   // DB820
{ S7_Optimized_Access := 'FALSE' }
VERSION : 0.1
BEGIN
END_DATA_BLOCK

DATA_BLOCK "ParAtd"   // DB830
TITLE = Parâmetros de Atuadores
{ S7_Optimized_Access := 'FALSE' }
VERSION : 0.1
BEGIN
END_DATA_BLOCK

DATA_BLOCK "ParEes"   // DB860
{ S7_Optimized_Access := 'FALSE' }
VERSION : 0.1
   VAR
      EES001_TamPec : Real;   // Selecionador de Peças - Tamanho da Peça (1P 2M 3G)
      EES001_PecMat : Real;   // Selecionador de Peças - Material da peça (Metal 1 ou plástico 2)
   END_VAR
BEGIN
END_DATA_BLOCK

// folder: (top level)

ORGANIZATION_BLOCK "Main"   // OB1, LAD, ProgramCycle
TITLE = "Main Program Sweep (Cycle)"
{ S7_Optimized_Access := 'TRUE' }
VERSION : 0.1
   VAR_INPUT
      Initial_Call : Bool;   // Initial call of this OB
      Remanence : Bool;   // =True, if remanent data are available
   END_VAR
   VAR_TEMP   // added for the SCL form of the ladder/FBD networks
      _w1 : Bool;
      _w2 : Bool;
      _w3 : Bool;
   END_VAR
BEGIN

REGION Network 1: ATUADORES
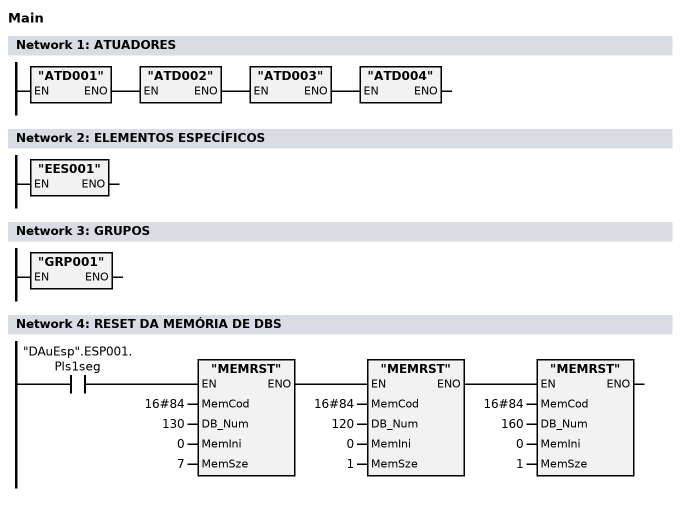
   RUNG wire#powerrail
      "ATD001"()
      "ATD002"()
      "ATD003"()
      "ATD004"()
   END_RUNG
   // the same network as SCL:
   "ATD001"(ENO => #_w1);
   "ATD002"(EN := #_w1, ENO => #_w2);
   "ATD003"(EN := #_w2, ENO => #_w3);
   IF #_w3 THEN "ATD004"(); END_IF;
END_REGION

REGION Network 2: ELEMENTOS ESPECÍFICOS
   RUNG wire#powerrail
      "EES001"()
   END_RUNG
   // the same network as SCL:
   "EES001"();
END_REGION

REGION Network 3: GRUPOS
   RUNG wire#powerrail
      "GRP001"()
   END_RUNG
   // the same network as SCL:
   "GRP001"();
END_REGION

REGION Network 4: RESET DA MEMÓRIA DE DBS
   RUNG wire#powerrail
      Contact( "DAuEsp".ESP001.Pls1seg )
      "MEMRST"(MemCod := 16#84, DB_Num := 130, MemIni := 0, MemSze := 7)
      "MEMRST"(MemCod := 16#84, DB_Num := 120, MemIni := 0, MemSze := 1)
      "MEMRST"(MemCod := 16#84, DB_Num := 160, MemIni := 0, MemSze := 1)
   END_RUNG
   // the same network as SCL:
   "MEMRST"(EN := "DAuEsp".ESP001.Pls1seg,
            MemCod := 16#84,
            DB_Num := 130,
            MemIni := 0,
            MemSze := 7,
            ENO => #_w1);
   "MEMRST"(EN := #_w1, MemCod := 16#84, DB_Num := 120, MemIni := 0, MemSze := 1, ENO => #_w2);
   IF #_w2 THEN "MEMRST"(MemCod := 16#84, DB_Num := 160, MemIni := 0, MemSze := 1); END_IF;
END_REGION
END_ORGANIZATION_BLOCK

// folder: FUNÇÕES

FUNCTION "MEMRST" : Void   // FC7, SCL
TITLE = Zeramento de áreas de memória
{ S7_Optimized_Access := 'TRUE' }
AUTHOR : Dimitri
FAMILY : UFLA
NAME : DEG
VERSION : 1.0
   VAR_INPUT
      MemCod : Byte;   // Código da área de memória (16#81=I 16#82=Q 16#83=M 16#84=DB)
      DB_Num : Int;   // Número do DB (deve ser zero para as áreas I, Q ou M)
      MemIni : Int;   // Byte inicial da área de memória a ser zerada
      MemSze : Int;   // Quantidade de bytes a serem zerados a partir do início indicado
   END_VAR
   VAR_TEMP
      i01Aux : Int;   // Auxiliar inteiro 01
   END_VAR
BEGIN
   // loop de zeramento
   IF #MemIni >= 0 AND #MemSze > 0 THEN
       FOR #i01Aux := #MemIni TO (#MemIni + #MemSze - 1) DO
           POKE(area := #MemCod,
                dbNumber := #DB_Num,
                byteOffset := #i01Aux,
                value := b#0);
       END_FOR;
   END_IF;
END_FUNCTION

FUNCTION "DMXCMD" : Void   // FC8, SCL
TITLE = Demultiplexação de comandos
{ S7_Optimized_Access := 'TRUE' }
AUTHOR : Dimitri
FAMILY : UFLA
NAME : DEG
VERSION : 3.0
   VAR_IN_OUT
      DmxFrm : DWord;   // Frame a ser demultiplexado
   END_VAR
   VAR_TEMP
      BlkNum : DInt;   // Número do "data block"
      BteNum : DInt;   // Número do byte
      BitNum : Int;   // Número do bit
   END_VAR
BEGIN
   IF #DmxFrm <> 0 THEN

       // decomposição do frame: block (14 bits) + byte (14 bits) + bit (4 bits)
       #BlkNum := DWORD_TO_DINT(SHR(IN := #DmxFrm, N := 18));
       #BteNum := DWORD_TO_DINT(SHR(IN := #DmxFrm, N := 4) AND DW#16383);
       #BitNum := DWORD_TO_INT(#DmxFrm AND DW#15);

       // zeramento do frame
       #DmxFrm := 0;

       // ajuste para acesso ao próximo byte
       IF #BitNum > 7 THEN
           #BteNum := #BteNum + 1;
           #BitNum := #BitNum - 8;
       END_IF;

       // aplicação do comando
       IF #BlkNum = 0 THEN
           POKE_BOOL(area := 16#83,
                     dbNumber := 0,
                     byteOffset := #BteNum,
                     bitOffset := #BitNum,
                     value := true); // comando na área M
       ELSE
           POKE_BOOL(area := 16#84,
                     dbNumber := #BlkNum,
                     byteOffset := #BteNum,
                     bitOffset := #BitNum,
                     value := true); // comando em data block
       END_IF;

   END_IF;
END_FUNCTION

FUNCTION "DEFPEC" : Void   // FC9, LAD
TITLE = Função que define qual peça está em transporte na esteira
{ S7_Optimized_Access := 'TRUE' }
VERSION : 0.1
   VAR_TEMP
      Aux : Bool;   // Auxiliar para
   END_VAR
   VAR_TEMP   // added for the SCL form of the ladder/FBD networks
      _w1 : Bool;
   END_VAR
BEGIN

REGION Network 1: Reset parâmetros
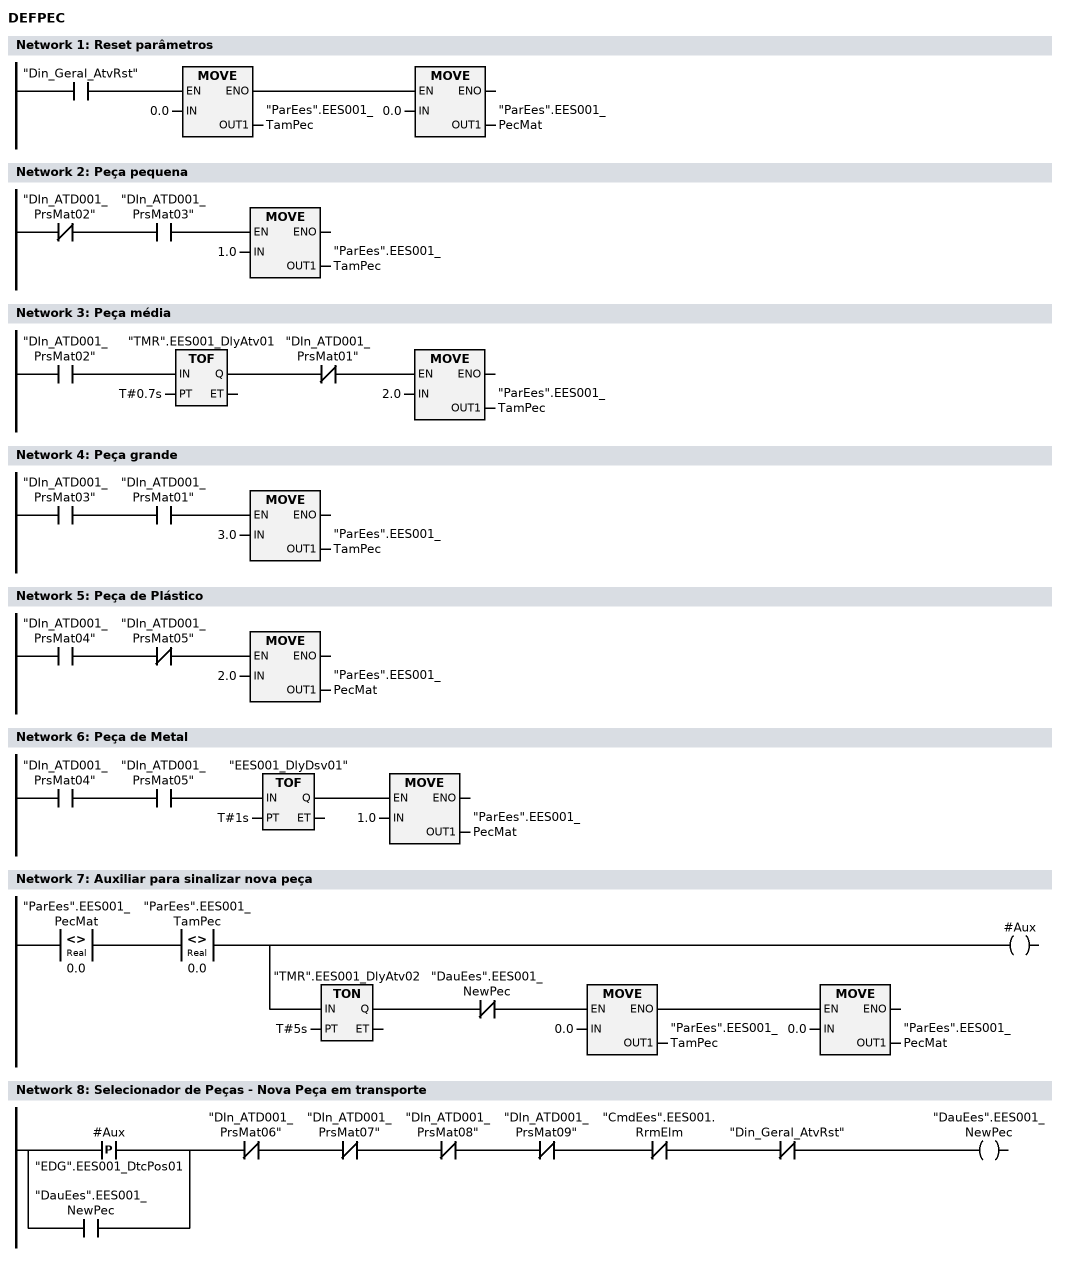
   RUNG wire#powerrail
      Contact( "Din_Geral_AtvRst" )
      Move(in := 0.0, out1 => "ParEes".EES001_TamPec)
      Move(in := 0.0, out1 => "ParEes".EES001_PecMat)
   END_RUNG
   // the same network as SCL:
   IF "Din_Geral_AtvRst" THEN
       "ParEes".EES001_TamPec := 0.0;
       "ParEes".EES001_PecMat := 0.0;
   END_IF;
END_REGION

REGION Network 2: Peça pequena
   RUNG wire#powerrail
      I_Contact( "DIn_ATD001_PrsMat02" )
      Contact( "DIn_ATD001_PrsMat03" )
      Move(in := 1.0, out1 => "ParEes".EES001_TamPec)
   END_RUNG
   // the same network as SCL:
   IF NOT "DIn_ATD001_PrsMat02" AND "DIn_ATD001_PrsMat03" THEN "ParEes".EES001_TamPec := 1.0; END_IF;
END_REGION

REGION Network 3: Peça média
   "TMR".EES001_DlyAtv01.TOF(IN := "DIn_ATD001_PrsMat02", PT := T#0.7s);
   IF "TMR".EES001_DlyAtv01.Q AND NOT "DIn_ATD001_PrsMat01" THEN "ParEes".EES001_TamPec := 2.0; END_IF;
END_REGION

REGION Network 4: Peça grande
   RUNG wire#powerrail
      Contact( "DIn_ATD001_PrsMat03" )
      Contact( "DIn_ATD001_PrsMat01" )
      Move(in := 3.0, out1 => "ParEes".EES001_TamPec)
   END_RUNG
   // the same network as SCL:
   IF "DIn_ATD001_PrsMat03" AND "DIn_ATD001_PrsMat01" THEN "ParEes".EES001_TamPec := 3.0; END_IF;
END_REGION

REGION Network 5: Peça de Plástico
   RUNG wire#powerrail
      Contact( "DIn_ATD001_PrsMat04" )
      I_Contact( "DIn_ATD001_PrsMat05" )
      Move(in := 2.0, out1 => "ParEes".EES001_PecMat)
   END_RUNG
   // the same network as SCL:
   IF "DIn_ATD001_PrsMat04" AND NOT "DIn_ATD001_PrsMat05" THEN "ParEes".EES001_PecMat := 2.0; END_IF;
END_REGION

REGION Network 6: Peça de Metal
   "EES001_DlyDsv01".TOF(IN := "DIn_ATD001_PrsMat04" AND "DIn_ATD001_PrsMat05", PT := T#1s);
   IF "EES001_DlyDsv01".Q THEN "ParEes".EES001_PecMat := 1.0; END_IF;
END_REGION

REGION Network 7: Auxiliar para sinalizar nova peça
   #Aux := ("ParEes".EES001_PecMat <> 0.0) AND ("ParEes".EES001_TamPec <> 0.0);
   "TMR".EES001_DlyAtv02.TON(IN := #Aux, PT := T#5s);
   IF "TMR".EES001_DlyAtv02.Q AND NOT "DauEes".EES001_NewPec THEN
       "ParEes".EES001_TamPec := 0.0;
       "ParEes".EES001_PecMat := 0.0;
   END_IF;
END_REGION

REGION Network 8: Selecionador de Peças - Nova Peça em transporte
   RUNG wire#powerrail
      P_Contact(operand := #Aux, bit := "EDG".EES001_DtcPos01)
      wire#w1
      I_Contact( "DIn_ATD001_PrsMat06" )
      I_Contact( "DIn_ATD001_PrsMat07" )
      I_Contact( "DIn_ATD001_PrsMat08" )
      I_Contact( "DIn_ATD001_PrsMat09" )
      I_Contact( "CmdEes".EES001.RrmElm )
      I_Contact( "Din_Geral_AtvRst" )
      Coil( "DauEes".EES001_NewPec )
   END_RUNG
   RUNG wire#powerrail
      Contact( "DauEes".EES001_NewPec )
   END_RUNG wire#w1
   // the same network as SCL:
   #_w1 := #Aux AND NOT "EDG".EES001_DtcPos01;   // rising edge of #Aux
   "EDG".EES001_DtcPos01 := #Aux;
   "DauEes".EES001_NewPec := (#_w1 OR "DauEes".EES001_NewPec) AND NOT "DIn_ATD001_PrsMat06" AND NOT "DIn_ATD001_PrsMat07" AND NOT "DIn_ATD001_PrsMat08" AND NOT "DIn_ATD001_PrsMat09" AND NOT "CmdEes".EES001.RrmElm AND NOT "Din_Geral_AtvRst";
END_REGION
END_FUNCTION

// folder: SUBROTINAS

FUNCTION "ATD001" : Void   // FC1, LAD
TITLE = Esteira Transportadora (ET-111)
{ S7_Optimized_Access := 'TRUE' }
VERSION : 0.1
BEGIN

REGION Network 1: Interlock - Condição de Emergência ativada
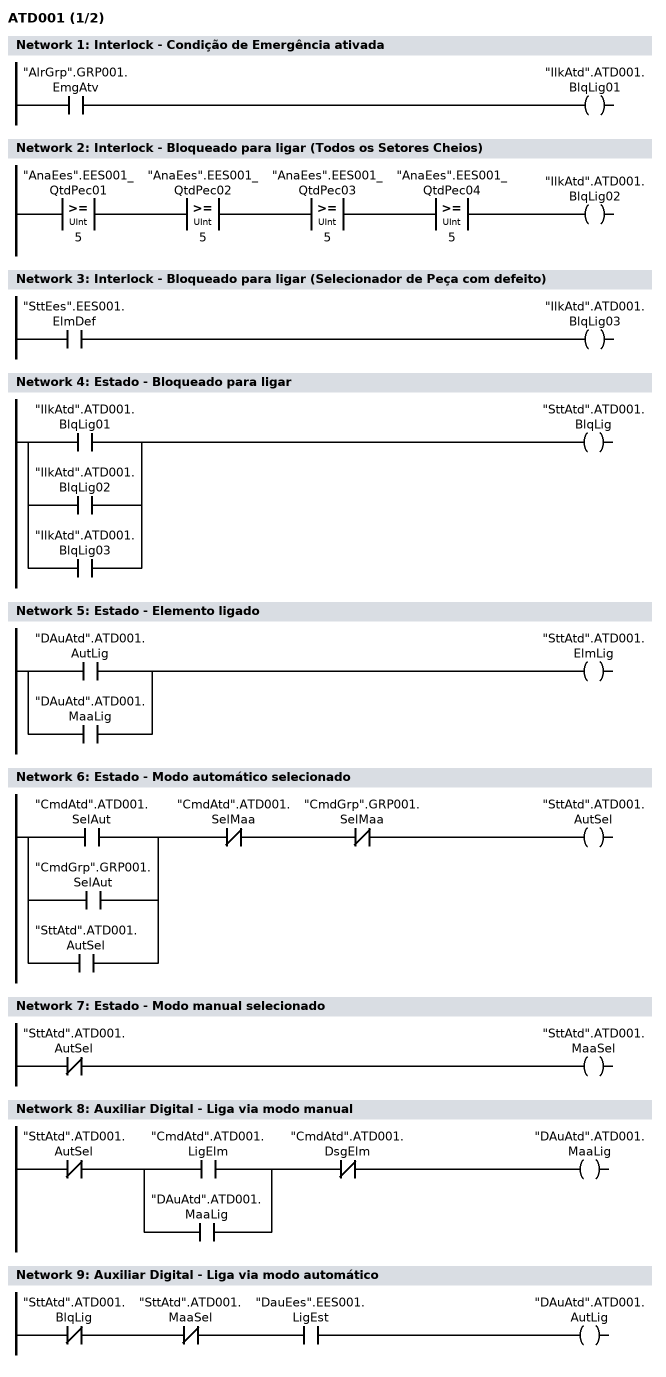
   RUNG wire#powerrail
      Contact( "AlrGrp".GRP001.EmgAtv )
      Coil( "IlkAtd".ATD001.BlqLig01 )
   END_RUNG
   // the same network as SCL:
   "IlkAtd".ATD001.BlqLig01 := "AlrGrp".GRP001.EmgAtv;
END_REGION

REGION Network 2: Interlock - Bloqueado para ligar (Todos os Setores Cheios)
   RUNG wire#powerrail
      { S7_Templates := "SrcType := UInt" } GE_Contact(in1 := "AnaEes".EES001_QtdPec01, in2 := 5)
      { S7_Templates := "SrcType := UInt" } GE_Contact(in1 := "AnaEes".EES001_QtdPec02, in2 := 5)
      { S7_Templates := "SrcType := UInt" } GE_Contact(in1 := "AnaEes".EES001_QtdPec03, in2 := 5)
      { S7_Templates := "SrcType := UInt" } GE_Contact(in1 := "AnaEes".EES001_QtdPec04, in2 := 5)
      Coil( "IlkAtd".ATD001.BlqLig02 )
   END_RUNG
   // the same network as SCL:
   "IlkAtd".ATD001.BlqLig02 := ("AnaEes".EES001_QtdPec01 >= 5) AND ("AnaEes".EES001_QtdPec02 >= 5) AND ("AnaEes".EES001_QtdPec03 >= 5) AND ("AnaEes".EES001_QtdPec04 >= 5);
END_REGION

REGION Network 3: Interlock - Bloqueado para ligar (Selecionador de Peça com defeito)
   RUNG wire#powerrail
      Contact( "SttEes".EES001.ElmDef )
      Coil( "IlkAtd".ATD001.BlqLig03 )
   END_RUNG
   // the same network as SCL:
   "IlkAtd".ATD001.BlqLig03 := "SttEes".EES001.ElmDef;
END_REGION

REGION Network 4: Estado - Bloqueado para ligar
   RUNG wire#powerrail
      Contact( "IlkAtd".ATD001.BlqLig01 )
      wire#w1
      Coil( "SttAtd".ATD001.BlqLig )
   END_RUNG
   RUNG wire#powerrail
      Contact( "IlkAtd".ATD001.BlqLig02 )
   END_RUNG wire#w1
   RUNG wire#powerrail
      Contact( "IlkAtd".ATD001.BlqLig03 )
   END_RUNG wire#w1
   // the same network as SCL:
   "SttAtd".ATD001.BlqLig := "IlkAtd".ATD001.BlqLig01 OR "IlkAtd".ATD001.BlqLig02 OR "IlkAtd".ATD001.BlqLig03;
END_REGION

REGION Network 5: Estado - Elemento ligado
   RUNG wire#powerrail
      Contact( "DAuAtd".ATD001.AutLig )
      wire#w1
      Coil( "SttAtd".ATD001.ElmLig )
   END_RUNG
   RUNG wire#powerrail
      Contact( "DAuAtd".ATD001.MaaLig )
   END_RUNG wire#w1
   // the same network as SCL:
   "SttAtd".ATD001.ElmLig := "DAuAtd".ATD001.AutLig OR "DAuAtd".ATD001.MaaLig;
END_REGION

REGION Network 6: Estado - Modo automático selecionado
   RUNG wire#powerrail
      Contact( "CmdAtd".ATD001.SelAut )
      wire#w1
      I_Contact( "CmdAtd".ATD001.SelMaa )
      I_Contact( "CmdGrp".GRP001.SelMaa )
      Coil( "SttAtd".ATD001.AutSel )
   END_RUNG
   RUNG wire#powerrail
      Contact( "CmdGrp".GRP001.SelAut )
   END_RUNG wire#w1
   RUNG wire#powerrail
      Contact( "SttAtd".ATD001.AutSel )
   END_RUNG wire#w1
   // the same network as SCL:
   "SttAtd".ATD001.AutSel := ("CmdAtd".ATD001.SelAut OR "CmdGrp".GRP001.SelAut OR "SttAtd".ATD001.AutSel) AND NOT "CmdAtd".ATD001.SelMaa AND NOT "CmdGrp".GRP001.SelMaa;
END_REGION

REGION Network 7: Estado - Modo manual selecionado
   RUNG wire#powerrail
      I_Contact( "SttAtd".ATD001.AutSel )
      Coil( "SttAtd".ATD001.MaaSel )
   END_RUNG
   // the same network as SCL:
   "SttAtd".ATD001.MaaSel := NOT "SttAtd".ATD001.AutSel;
END_REGION

REGION Network 8: Auxiliar Digital - Liga via modo manual
   RUNG wire#powerrail
      I_Contact( "SttAtd".ATD001.AutSel )
      wire#w1
      Contact( "CmdAtd".ATD001.LigElm )
      wire#w2
      I_Contact( "CmdAtd".ATD001.DsgElm )
      Coil( "DAuAtd".ATD001.MaaLig )
   END_RUNG
   RUNG wire#w1
      Contact( "DAuAtd".ATD001.MaaLig )
   END_RUNG wire#w2
   // the same network as SCL:
   "DAuAtd".ATD001.MaaLig := NOT "SttAtd".ATD001.AutSel AND ("CmdAtd".ATD001.LigElm OR "DAuAtd".ATD001.MaaLig) AND NOT "CmdAtd".ATD001.DsgElm;
END_REGION

REGION Network 9: Auxiliar Digital - Liga via modo automático
   RUNG wire#powerrail
      I_Contact( "SttAtd".ATD001.BlqLig )
      I_Contact( "SttAtd".ATD001.MaaSel )
      Contact( "DauEes".EES001.LigEst )
      Coil( "DAuAtd".ATD001.AutLig )
   END_RUNG
   // the same network as SCL:
   "DAuAtd".ATD001.AutLig := NOT "SttAtd".ATD001.BlqLig AND NOT "SttAtd".ATD001.MaaSel AND "DauEes".EES001.LigEst;
END_REGION

REGION Network 10: Saída Digital - Liga elemento
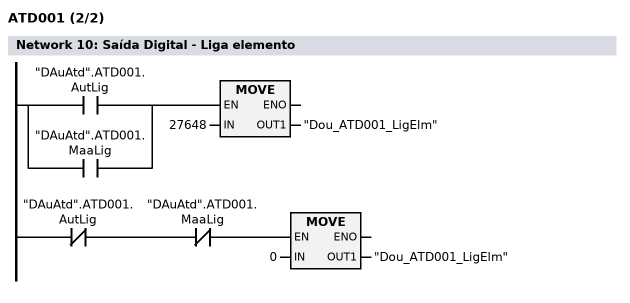
   RUNG wire#powerrail
      Contact( "DAuAtd".ATD001.AutLig )
      wire#w1
      Move(in := 27648, out1 => "Dou_ATD001_LigElm")
   END_RUNG
   RUNG wire#powerrail
      Contact( "DAuAtd".ATD001.MaaLig )
   END_RUNG wire#w1
   RUNG wire#powerrail
      I_Contact( "DAuAtd".ATD001.AutLig )
      I_Contact( "DAuAtd".ATD001.MaaLig )
      Move(in := 0, out1 => "Dou_ATD001_LigElm")
   END_RUNG
   // the same network as SCL:
   IF "DAuAtd".ATD001.AutLig OR "DAuAtd".ATD001.MaaLig THEN "Dou_ATD001_LigElm" := 27648; END_IF;
   IF NOT "DAuAtd".ATD001.AutLig AND NOT "DAuAtd".ATD001.MaaLig THEN "Dou_ATD001_LigElm" := 0; END_IF;
END_REGION
END_FUNCTION

FUNCTION "ATD002" : Void   // FC2, LAD
TITLE = Pistão Separador A (PI-111)
{ S7_Optimized_Access := 'TRUE' }
VERSION : 0.1
BEGIN

REGION Network 1: Interlock - Condição de Emergência ativada
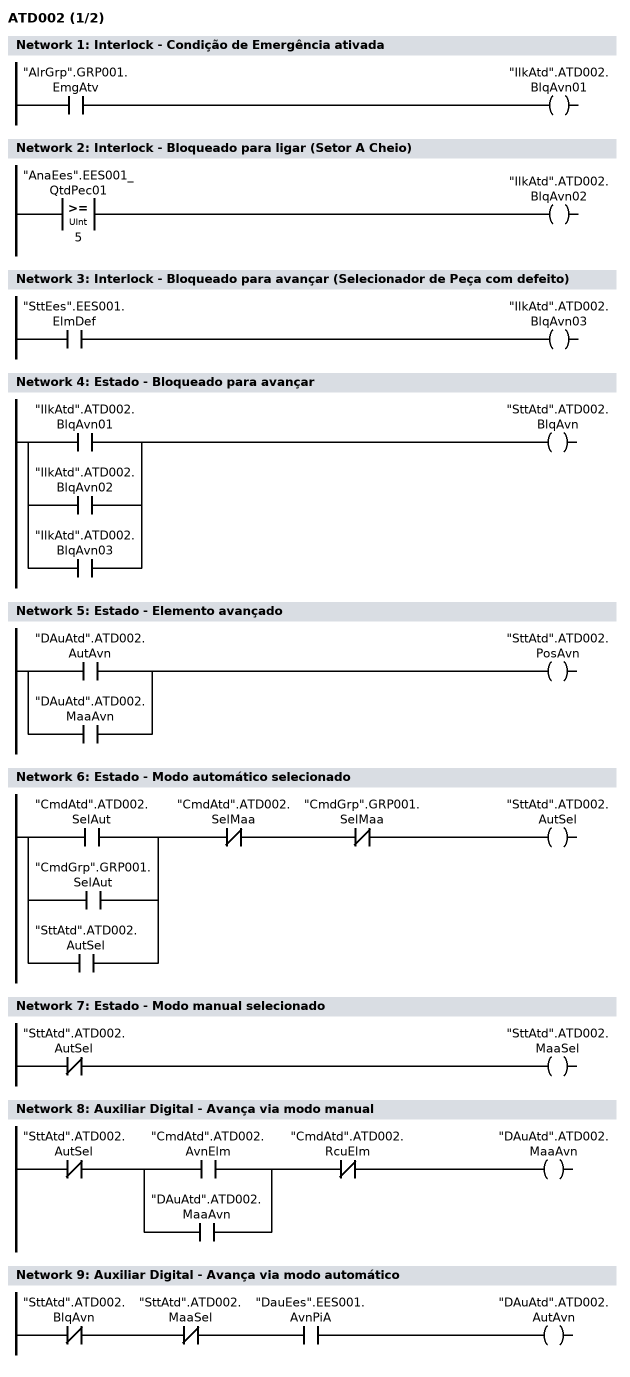
   RUNG wire#powerrail
      Contact( "AlrGrp".GRP001.EmgAtv )
      Coil( "IlkAtd".ATD002.BlqAvn01 )
   END_RUNG
   // the same network as SCL:
   "IlkAtd".ATD002.BlqAvn01 := "AlrGrp".GRP001.EmgAtv;
END_REGION

REGION Network 2: Interlock - Bloqueado para ligar (Setor A Cheio)
   RUNG wire#powerrail
      { S7_Templates := "SrcType := UInt" } GE_Contact(in1 := "AnaEes".EES001_QtdPec01, in2 := 5)
      Coil( "IlkAtd".ATD002.BlqAvn02 )
   END_RUNG
   // the same network as SCL:
   "IlkAtd".ATD002.BlqAvn02 := "AnaEes".EES001_QtdPec01 >= 5;
END_REGION

REGION Network 3: Interlock - Bloqueado para avançar (Selecionador de Peça com defeito)
   RUNG wire#powerrail
      Contact( "SttEes".EES001.ElmDef )
      Coil( "IlkAtd".ATD002.BlqAvn03 )
   END_RUNG
   // the same network as SCL:
   "IlkAtd".ATD002.BlqAvn03 := "SttEes".EES001.ElmDef;
END_REGION

REGION Network 4: Estado - Bloqueado para avançar
   RUNG wire#powerrail
      Contact( "IlkAtd".ATD002.BlqAvn01 )
      wire#w1
      Coil( "SttAtd".ATD002.BlqAvn )
   END_RUNG
   RUNG wire#powerrail
      Contact( "IlkAtd".ATD002.BlqAvn02 )
   END_RUNG wire#w1
   RUNG wire#powerrail
      Contact( "IlkAtd".ATD002.BlqAvn03 )
   END_RUNG wire#w1
   // the same network as SCL:
   "SttAtd".ATD002.BlqAvn := "IlkAtd".ATD002.BlqAvn01 OR "IlkAtd".ATD002.BlqAvn02 OR "IlkAtd".ATD002.BlqAvn03;
END_REGION

REGION Network 5: Estado - Elemento avançado
   RUNG wire#powerrail
      Contact( "DAuAtd".ATD002.AutAvn )
      wire#w1
      Coil( "SttAtd".ATD002.PosAvn )
   END_RUNG
   RUNG wire#powerrail
      Contact( "DAuAtd".ATD002.MaaAvn )
   END_RUNG wire#w1
   // the same network as SCL:
   "SttAtd".ATD002.PosAvn := "DAuAtd".ATD002.AutAvn OR "DAuAtd".ATD002.MaaAvn;
END_REGION

REGION Network 6: Estado - Modo automático selecionado
   RUNG wire#powerrail
      Contact( "CmdAtd".ATD002.SelAut )
      wire#w1
      I_Contact( "CmdAtd".ATD002.SelMaa )
      I_Contact( "CmdGrp".GRP001.SelMaa )
      Coil( "SttAtd".ATD002.AutSel )
   END_RUNG
   RUNG wire#powerrail
      Contact( "CmdGrp".GRP001.SelAut )
   END_RUNG wire#w1
   RUNG wire#powerrail
      Contact( "SttAtd".ATD002.AutSel )
   END_RUNG wire#w1
   // the same network as SCL:
   "SttAtd".ATD002.AutSel := ("CmdAtd".ATD002.SelAut OR "CmdGrp".GRP001.SelAut OR "SttAtd".ATD002.AutSel) AND NOT "CmdAtd".ATD002.SelMaa AND NOT "CmdGrp".GRP001.SelMaa;
END_REGION

REGION Network 7: Estado - Modo manual selecionado
   RUNG wire#powerrail
      I_Contact( "SttAtd".ATD002.AutSel )
      Coil( "SttAtd".ATD002.MaaSel )
   END_RUNG
   // the same network as SCL:
   "SttAtd".ATD002.MaaSel := NOT "SttAtd".ATD002.AutSel;
END_REGION

REGION Network 8: Auxiliar Digital - Avança via modo manual
   RUNG wire#powerrail
      I_Contact( "SttAtd".ATD002.AutSel )
      wire#w1
      Contact( "CmdAtd".ATD002.AvnElm )
      wire#w2
      I_Contact( "CmdAtd".ATD002.RcuElm )
      Coil( "DAuAtd".ATD002.MaaAvn )
   END_RUNG
   RUNG wire#w1
      Contact( "DAuAtd".ATD002.MaaAvn )
   END_RUNG wire#w2
   // the same network as SCL:
   "DAuAtd".ATD002.MaaAvn := NOT "SttAtd".ATD002.AutSel AND ("CmdAtd".ATD002.AvnElm OR "DAuAtd".ATD002.MaaAvn) AND NOT "CmdAtd".ATD002.RcuElm;
END_REGION

REGION Network 9: Auxiliar Digital - Avança via modo automático
   RUNG wire#powerrail
      I_Contact( "SttAtd".ATD002.BlqAvn )
      I_Contact( "SttAtd".ATD002.MaaSel )
      Contact( "DauEes".EES001.AvnPiA )
      Coil( "DAuAtd".ATD002.AutAvn )
   END_RUNG
   // the same network as SCL:
   "DAuAtd".ATD002.AutAvn := NOT "SttAtd".ATD002.BlqAvn AND NOT "SttAtd".ATD002.MaaSel AND "DauEes".EES001.AvnPiA;
END_REGION

REGION Network 10: Saída Digital - Avança elemento
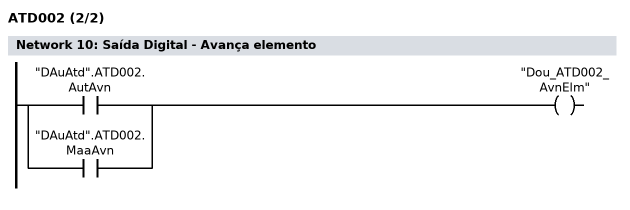
   RUNG wire#powerrail
      Contact( "DAuAtd".ATD002.AutAvn )
      wire#w1
      Coil( "Dou_ATD002_AvnElm" )
   END_RUNG
   RUNG wire#powerrail
      Contact( "DAuAtd".ATD002.MaaAvn )
   END_RUNG wire#w1
   // the same network as SCL:
   "Dou_ATD002_AvnElm" := "DAuAtd".ATD002.AutAvn OR "DAuAtd".ATD002.MaaAvn;
END_REGION
END_FUNCTION

FUNCTION "ATD003" : Void   // FC3, LAD
TITLE = Pistão Separador B (PI-112)
{ S7_Optimized_Access := 'TRUE' }
VERSION : 0.1
BEGIN

REGION Network 1: Interlock - Condição de Emergência ativada
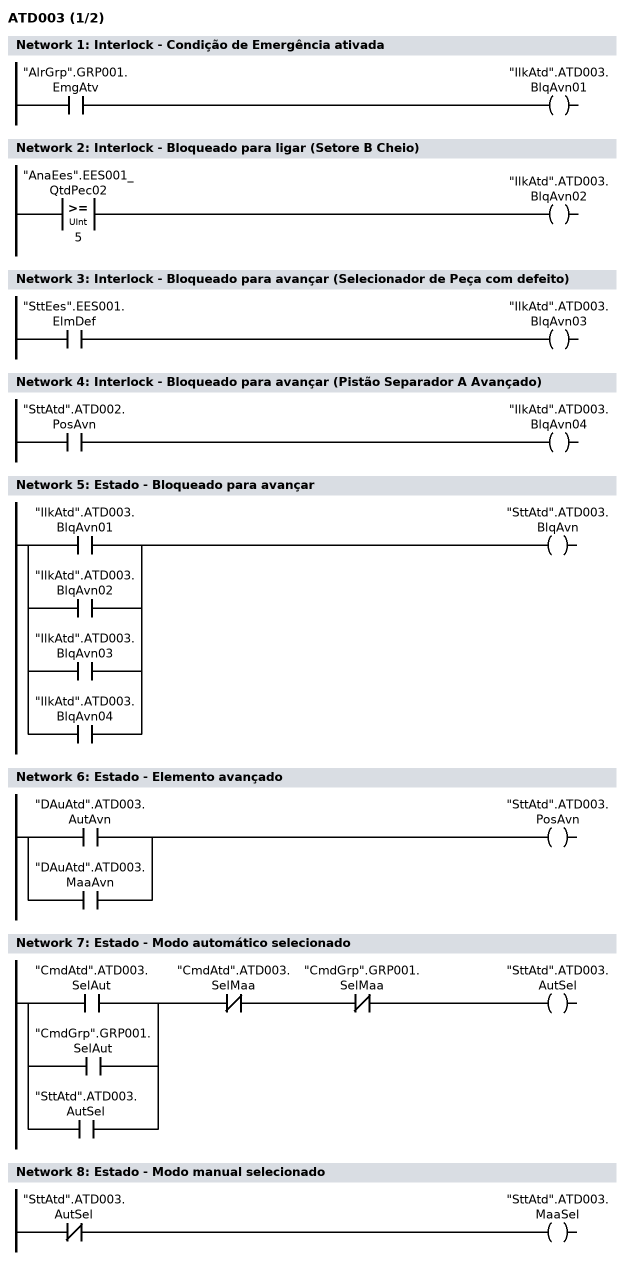
   RUNG wire#powerrail
      Contact( "AlrGrp".GRP001.EmgAtv )
      Coil( "IlkAtd".ATD003.BlqAvn01 )
   END_RUNG
   // the same network as SCL:
   "IlkAtd".ATD003.BlqAvn01 := "AlrGrp".GRP001.EmgAtv;
END_REGION

REGION Network 2: Interlock - Bloqueado para ligar (Setore B Cheio)
   RUNG wire#powerrail
      { S7_Templates := "SrcType := UInt" } GE_Contact(in1 := "AnaEes".EES001_QtdPec02, in2 := 5)
      Coil( "IlkAtd".ATD003.BlqAvn02 )
   END_RUNG
   // the same network as SCL:
   "IlkAtd".ATD003.BlqAvn02 := "AnaEes".EES001_QtdPec02 >= 5;
END_REGION

REGION Network 3: Interlock - Bloqueado para avançar (Selecionador de Peça com defeito)
   RUNG wire#powerrail
      Contact( "SttEes".EES001.ElmDef )
      Coil( "IlkAtd".ATD003.BlqAvn03 )
   END_RUNG
   // the same network as SCL:
   "IlkAtd".ATD003.BlqAvn03 := "SttEes".EES001.ElmDef;
END_REGION

REGION Network 4: Interlock - Bloqueado para avançar (Pistão Separador A Avançado)
   RUNG wire#powerrail
      Contact( "SttAtd".ATD002.PosAvn )
      Coil( "IlkAtd".ATD003.BlqAvn04 )
   END_RUNG
   // the same network as SCL:
   "IlkAtd".ATD003.BlqAvn04 := "SttAtd".ATD002.PosAvn;
END_REGION

REGION Network 5: Estado - Bloqueado para avançar
   RUNG wire#powerrail
      Contact( "IlkAtd".ATD003.BlqAvn01 )
      wire#w1
      Coil( "SttAtd".ATD003.BlqAvn )
   END_RUNG
   RUNG wire#powerrail
      Contact( "IlkAtd".ATD003.BlqAvn02 )
   END_RUNG wire#w1
   RUNG wire#powerrail
      Contact( "IlkAtd".ATD003.BlqAvn03 )
   END_RUNG wire#w1
   RUNG wire#powerrail
      Contact( "IlkAtd".ATD003.BlqAvn04 )
   END_RUNG wire#w1
   // the same network as SCL:
   "SttAtd".ATD003.BlqAvn := "IlkAtd".ATD003.BlqAvn01 OR "IlkAtd".ATD003.BlqAvn02 OR "IlkAtd".ATD003.BlqAvn03 OR "IlkAtd".ATD003.BlqAvn04;
END_REGION

REGION Network 6: Estado - Elemento avançado
   RUNG wire#powerrail
      Contact( "DAuAtd".ATD003.AutAvn )
      wire#w1
      Coil( "SttAtd".ATD003.PosAvn )
   END_RUNG
   RUNG wire#powerrail
      Contact( "DAuAtd".ATD003.MaaAvn )
   END_RUNG wire#w1
   // the same network as SCL:
   "SttAtd".ATD003.PosAvn := "DAuAtd".ATD003.AutAvn OR "DAuAtd".ATD003.MaaAvn;
END_REGION

REGION Network 7: Estado - Modo automático selecionado
   RUNG wire#powerrail
      Contact( "CmdAtd".ATD003.SelAut )
      wire#w1
      I_Contact( "CmdAtd".ATD003.SelMaa )
      I_Contact( "CmdGrp".GRP001.SelMaa )
      Coil( "SttAtd".ATD003.AutSel )
   END_RUNG
   RUNG wire#powerrail
      Contact( "CmdGrp".GRP001.SelAut )
   END_RUNG wire#w1
   RUNG wire#powerrail
      Contact( "SttAtd".ATD003.AutSel )
   END_RUNG wire#w1
   // the same network as SCL:
   "SttAtd".ATD003.AutSel := ("CmdAtd".ATD003.SelAut OR "CmdGrp".GRP001.SelAut OR "SttAtd".ATD003.AutSel) AND NOT "CmdAtd".ATD003.SelMaa AND NOT "CmdGrp".GRP001.SelMaa;
END_REGION

REGION Network 8: Estado - Modo manual selecionado
   RUNG wire#powerrail
      I_Contact( "SttAtd".ATD003.AutSel )
      Coil( "SttAtd".ATD003.MaaSel )
   END_RUNG
   // the same network as SCL:
   "SttAtd".ATD003.MaaSel := NOT "SttAtd".ATD003.AutSel;
END_REGION

REGION Network 9: Auxiliar Digital - Avança via modo manual
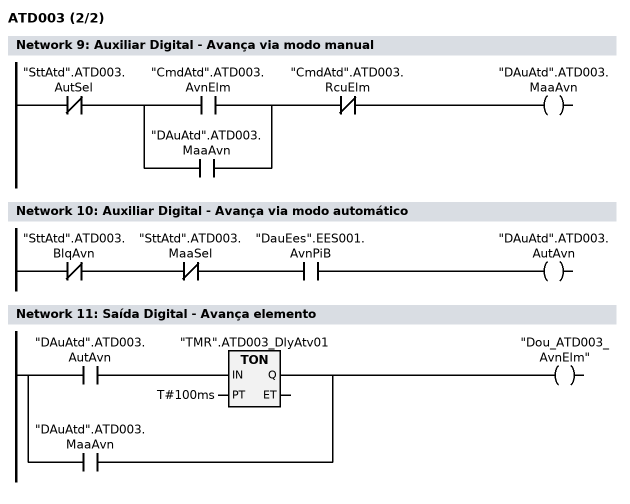
   RUNG wire#powerrail
      I_Contact( "SttAtd".ATD003.AutSel )
      wire#w1
      Contact( "CmdAtd".ATD003.AvnElm )
      wire#w2
      I_Contact( "CmdAtd".ATD003.RcuElm )
      Coil( "DAuAtd".ATD003.MaaAvn )
   END_RUNG
   RUNG wire#w1
      Contact( "DAuAtd".ATD003.MaaAvn )
   END_RUNG wire#w2
   // the same network as SCL:
   "DAuAtd".ATD003.MaaAvn := NOT "SttAtd".ATD003.AutSel AND ("CmdAtd".ATD003.AvnElm OR "DAuAtd".ATD003.MaaAvn) AND NOT "CmdAtd".ATD003.RcuElm;
END_REGION

REGION Network 10: Auxiliar Digital - Avança via modo automático
   RUNG wire#powerrail
      I_Contact( "SttAtd".ATD003.BlqAvn )
      I_Contact( "SttAtd".ATD003.MaaSel )
      Contact( "DauEes".EES001.AvnPiB )
      Coil( "DAuAtd".ATD003.AutAvn )
   END_RUNG
   // the same network as SCL:
   "DAuAtd".ATD003.AutAvn := NOT "SttAtd".ATD003.BlqAvn AND NOT "SttAtd".ATD003.MaaSel AND "DauEes".EES001.AvnPiB;
END_REGION

REGION Network 11: Saída Digital - Avança elemento
   "TMR".ATD003_DlyAtv01.TON(IN := "DAuAtd".ATD003.AutAvn, PT := T#100ms);
   "Dou_ATD003_AvnElm" := "TMR".ATD003_DlyAtv01.Q OR "DAuAtd".ATD003.MaaAvn;
END_REGION
END_FUNCTION

FUNCTION "ATD004" : Void   // FC4, LAD
TITLE = Pistão Separador C (PI-113)
{ S7_Optimized_Access := 'TRUE' }
VERSION : 0.1
BEGIN

REGION Network 1: Interlock - Condição de Emergência ativada
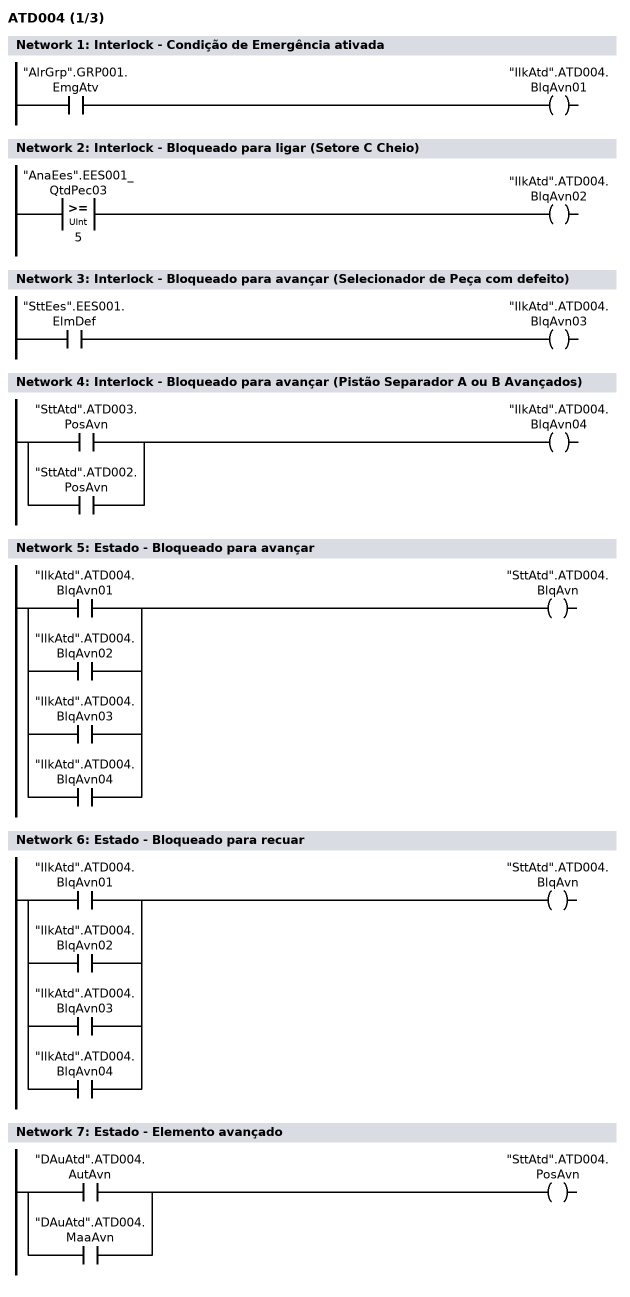
   RUNG wire#powerrail
      Contact( "AlrGrp".GRP001.EmgAtv )
      Coil( "IlkAtd".ATD004.BlqAvn01 )
   END_RUNG
   // the same network as SCL:
   "IlkAtd".ATD004.BlqAvn01 := "AlrGrp".GRP001.EmgAtv;
END_REGION

REGION Network 2: Interlock - Bloqueado para ligar (Setore C Cheio)
   RUNG wire#powerrail
      { S7_Templates := "SrcType := UInt" } GE_Contact(in1 := "AnaEes".EES001_QtdPec03, in2 := 5)
      Coil( "IlkAtd".ATD004.BlqAvn02 )
   END_RUNG
   // the same network as SCL:
   "IlkAtd".ATD004.BlqAvn02 := "AnaEes".EES001_QtdPec03 >= 5;
END_REGION

REGION Network 3: Interlock - Bloqueado para avançar (Selecionador de Peça com defeito)
   RUNG wire#powerrail
      Contact( "SttEes".EES001.ElmDef )
      Coil( "IlkAtd".ATD004.BlqAvn03 )
   END_RUNG
   // the same network as SCL:
   "IlkAtd".ATD004.BlqAvn03 := "SttEes".EES001.ElmDef;
END_REGION

REGION Network 4: Interlock - Bloqueado para avançar (Pistão Separador A ou B Avançados)
   RUNG wire#powerrail
      Contact( "SttAtd".ATD003.PosAvn )
      wire#w1
      Coil( "IlkAtd".ATD004.BlqAvn04 )
   END_RUNG
   RUNG wire#powerrail
      Contact( "SttAtd".ATD002.PosAvn )
   END_RUNG wire#w1
   // the same network as SCL:
   "IlkAtd".ATD004.BlqAvn04 := "SttAtd".ATD003.PosAvn OR "SttAtd".ATD002.PosAvn;
END_REGION

REGION Network 5: Estado - Bloqueado para avançar
   RUNG wire#powerrail
      Contact( "IlkAtd".ATD004.BlqAvn01 )
      wire#w1
      Coil( "SttAtd".ATD004.BlqAvn )
   END_RUNG
   RUNG wire#powerrail
      Contact( "IlkAtd".ATD004.BlqAvn02 )
   END_RUNG wire#w1
   RUNG wire#powerrail
      Contact( "IlkAtd".ATD004.BlqAvn03 )
   END_RUNG wire#w1
   RUNG wire#powerrail
      Contact( "IlkAtd".ATD004.BlqAvn04 )
   END_RUNG wire#w1
   // the same network as SCL:
   "SttAtd".ATD004.BlqAvn := "IlkAtd".ATD004.BlqAvn01 OR "IlkAtd".ATD004.BlqAvn02 OR "IlkAtd".ATD004.BlqAvn03 OR "IlkAtd".ATD004.BlqAvn04;
END_REGION

REGION Network 6: Estado - Bloqueado para recuar
   RUNG wire#powerrail
      Contact( "IlkAtd".ATD004.BlqAvn01 )
      wire#w1
      Coil( "SttAtd".ATD004.BlqAvn )
   END_RUNG
   RUNG wire#powerrail
      Contact( "IlkAtd".ATD004.BlqAvn02 )
   END_RUNG wire#w1
   RUNG wire#powerrail
      Contact( "IlkAtd".ATD004.BlqAvn03 )
   END_RUNG wire#w1
   RUNG wire#powerrail
      Contact( "IlkAtd".ATD004.BlqAvn04 )
   END_RUNG wire#w1
   // the same network as SCL:
   "SttAtd".ATD004.BlqAvn := "IlkAtd".ATD004.BlqAvn01 OR "IlkAtd".ATD004.BlqAvn02 OR "IlkAtd".ATD004.BlqAvn03 OR "IlkAtd".ATD004.BlqAvn04;
END_REGION

REGION Network 7: Estado - Elemento avançado
   RUNG wire#powerrail
      Contact( "DAuAtd".ATD004.AutAvn )
      wire#w1
      Coil( "SttAtd".ATD004.PosAvn )
   END_RUNG
   RUNG wire#powerrail
      Contact( "DAuAtd".ATD004.MaaAvn )
   END_RUNG wire#w1
   // the same network as SCL:
   "SttAtd".ATD004.PosAvn := "DAuAtd".ATD004.AutAvn OR "DAuAtd".ATD004.MaaAvn;
END_REGION

REGION Network 8: Estado - Elemento recuado
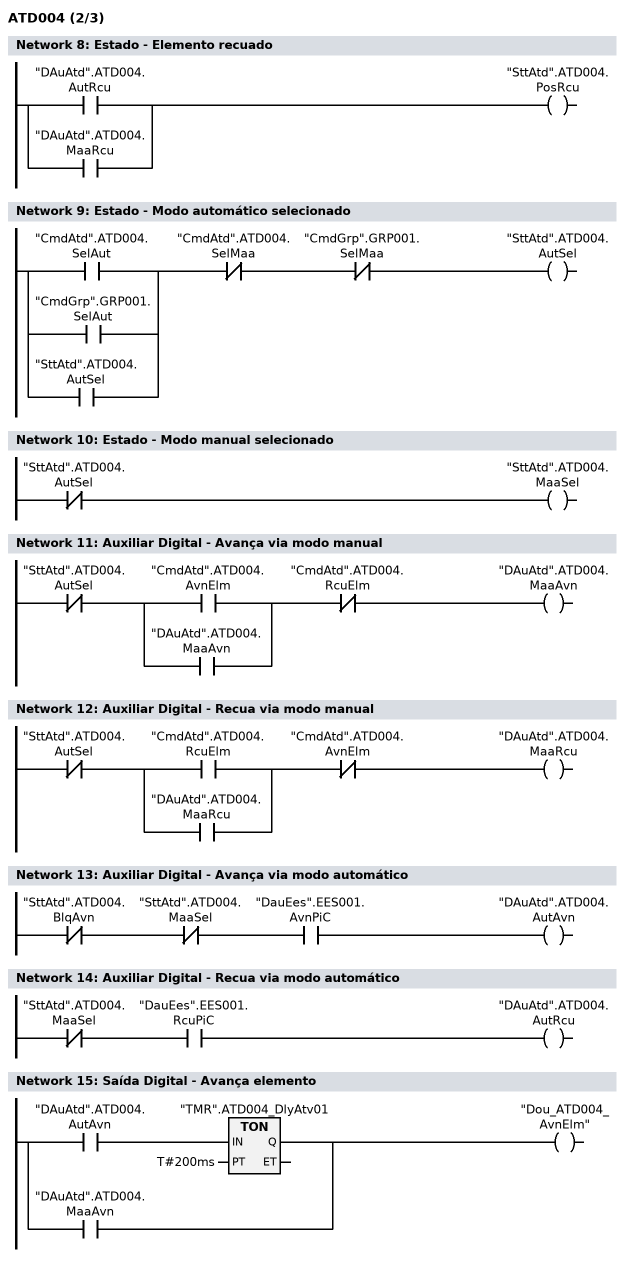
   RUNG wire#powerrail
      Contact( "DAuAtd".ATD004.AutRcu )
      wire#w1
      Coil( "SttAtd".ATD004.PosRcu )
   END_RUNG
   RUNG wire#powerrail
      Contact( "DAuAtd".ATD004.MaaRcu )
   END_RUNG wire#w1
   // the same network as SCL:
   "SttAtd".ATD004.PosRcu := "DAuAtd".ATD004.AutRcu OR "DAuAtd".ATD004.MaaRcu;
END_REGION

REGION Network 9: Estado - Modo automático selecionado
   RUNG wire#powerrail
      Contact( "CmdAtd".ATD004.SelAut )
      wire#w1
      I_Contact( "CmdAtd".ATD004.SelMaa )
      I_Contact( "CmdGrp".GRP001.SelMaa )
      Coil( "SttAtd".ATD004.AutSel )
   END_RUNG
   RUNG wire#powerrail
      Contact( "CmdGrp".GRP001.SelAut )
   END_RUNG wire#w1
   RUNG wire#powerrail
      Contact( "SttAtd".ATD004.AutSel )
   END_RUNG wire#w1
   // the same network as SCL:
   "SttAtd".ATD004.AutSel := ("CmdAtd".ATD004.SelAut OR "CmdGrp".GRP001.SelAut OR "SttAtd".ATD004.AutSel) AND NOT "CmdAtd".ATD004.SelMaa AND NOT "CmdGrp".GRP001.SelMaa;
END_REGION

REGION Network 10: Estado - Modo manual selecionado
   RUNG wire#powerrail
      I_Contact( "SttAtd".ATD004.AutSel )
      Coil( "SttAtd".ATD004.MaaSel )
   END_RUNG
   // the same network as SCL:
   "SttAtd".ATD004.MaaSel := NOT "SttAtd".ATD004.AutSel;
END_REGION

REGION Network 11: Auxiliar Digital - Avança via modo manual
   RUNG wire#powerrail
      I_Contact( "SttAtd".ATD004.AutSel )
      wire#w1
      Contact( "CmdAtd".ATD004.AvnElm )
      wire#w2
      I_Contact( "CmdAtd".ATD004.RcuElm )
      Coil( "DAuAtd".ATD004.MaaAvn )
   END_RUNG
   RUNG wire#w1
      Contact( "DAuAtd".ATD004.MaaAvn )
   END_RUNG wire#w2
   // the same network as SCL:
   "DAuAtd".ATD004.MaaAvn := NOT "SttAtd".ATD004.AutSel AND ("CmdAtd".ATD004.AvnElm OR "DAuAtd".ATD004.MaaAvn) AND NOT "CmdAtd".ATD004.RcuElm;
END_REGION

REGION Network 12: Auxiliar Digital - Recua via modo manual
   RUNG wire#powerrail
      I_Contact( "SttAtd".ATD004.AutSel )
      wire#w1
      Contact( "CmdAtd".ATD004.RcuElm )
      wire#w2
      I_Contact( "CmdAtd".ATD004.AvnElm )
      Coil( "DAuAtd".ATD004.MaaRcu )
   END_RUNG
   RUNG wire#w1
      Contact( "DAuAtd".ATD004.MaaRcu )
   END_RUNG wire#w2
   // the same network as SCL:
   "DAuAtd".ATD004.MaaRcu := NOT "SttAtd".ATD004.AutSel AND ("CmdAtd".ATD004.RcuElm OR "DAuAtd".ATD004.MaaRcu) AND NOT "CmdAtd".ATD004.AvnElm;
END_REGION

REGION Network 13: Auxiliar Digital - Avança via modo automático
   RUNG wire#powerrail
      I_Contact( "SttAtd".ATD004.BlqAvn )
      I_Contact( "SttAtd".ATD004.MaaSel )
      Contact( "DauEes".EES001.AvnPiC )
      Coil( "DAuAtd".ATD004.AutAvn )
   END_RUNG
   // the same network as SCL:
   "DAuAtd".ATD004.AutAvn := NOT "SttAtd".ATD004.BlqAvn AND NOT "SttAtd".ATD004.MaaSel AND "DauEes".EES001.AvnPiC;
END_REGION

REGION Network 14: Auxiliar Digital - Recua via modo automático
   RUNG wire#powerrail
      I_Contact( "SttAtd".ATD004.MaaSel )
      Contact( "DauEes".EES001.RcuPiC )
      Coil( "DAuAtd".ATD004.AutRcu )
   END_RUNG
   // the same network as SCL:
   "DAuAtd".ATD004.AutRcu := NOT "SttAtd".ATD004.MaaSel AND "DauEes".EES001.RcuPiC;
END_REGION

REGION Network 15: Saída Digital - Avança elemento
   "TMR".ATD004_DlyAtv01.TON(IN := "DAuAtd".ATD004.AutAvn, PT := T#200ms);
   "Dou_ATD004_AvnElm" := "TMR".ATD004_DlyAtv01.Q OR "DAuAtd".ATD004.MaaAvn;
END_REGION

REGION Network 16: Saída Digital - Recua elemento
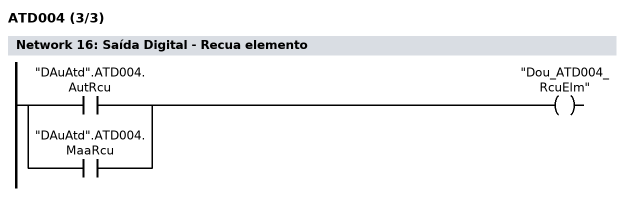
   RUNG wire#powerrail
      Contact( "DAuAtd".ATD004.AutRcu )
      wire#w1
      Coil( "Dou_ATD004_RcuElm" )
   END_RUNG
   RUNG wire#powerrail
      Contact( "DAuAtd".ATD004.MaaRcu )
   END_RUNG wire#w1
   // the same network as SCL:
   "Dou_ATD004_RcuElm" := "DAuAtd".ATD004.AutRcu OR "DAuAtd".ATD004.MaaRcu;
END_REGION
END_FUNCTION

FUNCTION "GRP001" : Void   // FC5, LAD
TITLE = Geral
{ S7_Optimized_Access := 'TRUE' }
VERSION : 0.1
   VAR_TEMP   // added for the SCL form of the ladder/FBD networks
      _w1 : Bool;
   END_VAR
BEGIN

REGION Network 1: Geral - Condição de Emergência Ativada
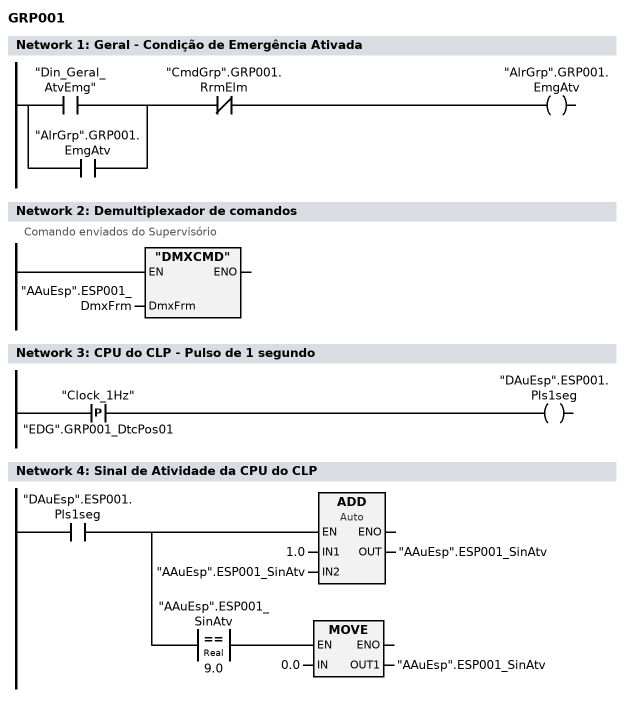
   RUNG wire#powerrail
      Contact( "Din_Geral_AtvEmg" )
      wire#w1
      I_Contact( "CmdGrp".GRP001.RrmElm )
      Coil( "AlrGrp".GRP001.EmgAtv )
   END_RUNG
   RUNG wire#powerrail
      Contact( "AlrGrp".GRP001.EmgAtv )
   END_RUNG wire#w1
   // the same network as SCL:
   "AlrGrp".GRP001.EmgAtv := ("Din_Geral_AtvEmg" OR "AlrGrp".GRP001.EmgAtv) AND NOT "CmdGrp".GRP001.RrmElm;
END_REGION

REGION Network 2: Demultiplexador de comandos
   // Comando enviados do Supervisório
   RUNG wire#powerrail
      "DMXCMD"(DmxFrm := "AAuEsp".ESP001_DmxFrm)
   END_RUNG
   // the same network as SCL:
   "DMXCMD"(DmxFrm := "AAuEsp".ESP001_DmxFrm);
END_REGION

REGION Network 3: CPU do CLP - Pulso de 1 segundo
   RUNG wire#powerrail
      P_Contact(operand := "Clock_1Hz", bit := "EDG".GRP001_DtcPos01)
      Coil( "DAuEsp".ESP001.Pls1seg )
   END_RUNG
   // the same network as SCL:
   #_w1 := "Clock_1Hz" AND NOT "EDG".GRP001_DtcPos01;   // rising edge of "Clock_1Hz"
   "EDG".GRP001_DtcPos01 := "Clock_1Hz";
   "DAuEsp".ESP001.Pls1seg := #_w1;
END_REGION

REGION Network 4: Sinal de Atividade da CPU do CLP
   RUNG wire#powerrail
      Contact( "DAuEsp".ESP001.Pls1seg )
      wire#w1
      Add(in1 := 1.0, in2 := "AAuEsp".ESP001_SinAtv, out => "AAuEsp".ESP001_SinAtv)
   END_RUNG
   RUNG wire#w1
      { S7_Templates := "SrcType := Real" } EQ_Contact(in1 := "AAuEsp".ESP001_SinAtv, in2 := 9.0)
      Move(in := 0.0, out1 => "AAuEsp".ESP001_SinAtv)
   END_RUNG
   // the same network as SCL:
   IF "DAuEsp".ESP001.Pls1seg THEN "AAuEsp".ESP001_SinAtv := 1.0 + "AAuEsp".ESP001_SinAtv; END_IF;
   IF "DAuEsp".ESP001.Pls1seg AND ("AAuEsp".ESP001_SinAtv = 9.0) THEN "AAuEsp".ESP001_SinAtv := 0.0; END_IF;
END_REGION
END_FUNCTION

FUNCTION "EES001" : Void   // FC6, LAD
TITLE = Selecionador de Peças
{ S7_Optimized_Access := 'TRUE' }
VERSION : 0.1
   VAR_TEMP
      Aux : Bool;   // Auxiliar para Recuar Pistão C
      Tempo_Transporte : Time;   // Auxiliar para marcar tempo em transporte
   END_VAR
   VAR_TEMP   // added for the SCL form of the ladder/FBD networks
      _w1 : Bool;
   END_VAR
BEGIN

REGION Network 1: Alarme - Limite Excedido (Mais de uma peça em transporte)
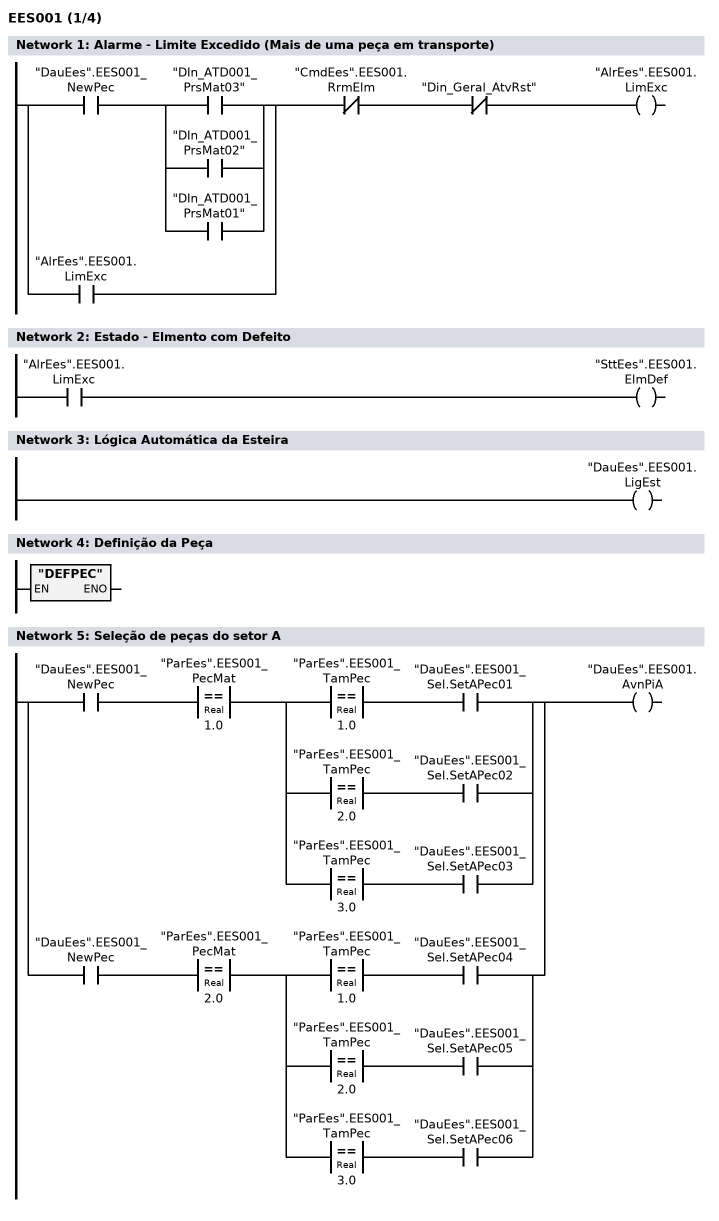
   RUNG wire#powerrail
      Contact( "DauEes".EES001_NewPec )
      wire#w1
      Contact( "DIn_ATD001_PrsMat03" )
      wire#w2
      I_Contact( "CmdEes".EES001.RrmElm )
      I_Contact( "Din_Geral_AtvRst" )
      Coil( "AlrEes".EES001.LimExc )
   END_RUNG
   RUNG wire#w1
      Contact( "DIn_ATD001_PrsMat02" )
   END_RUNG wire#w2
   RUNG wire#w1
      Contact( "DIn_ATD001_PrsMat01" )
   END_RUNG wire#w2
   RUNG wire#powerrail
      Contact( "AlrEes".EES001.LimExc )
   END_RUNG wire#w2
   // the same network as SCL:
   "AlrEes".EES001.LimExc := (("DauEes".EES001_NewPec AND ("DIn_ATD001_PrsMat03" OR "DIn_ATD001_PrsMat02" OR "DIn_ATD001_PrsMat01")) OR "AlrEes".EES001.LimExc) AND NOT "CmdEes".EES001.RrmElm AND NOT "Din_Geral_AtvRst";
END_REGION

REGION Network 2: Estado - Elmento com Defeito
   RUNG wire#powerrail
      Contact( "AlrEes".EES001.LimExc )
      Coil( "SttEes".EES001.ElmDef )
   END_RUNG
   // the same network as SCL:
   "SttEes".EES001.ElmDef := "AlrEes".EES001.LimExc;
END_REGION

REGION Network 3: Lógica Automática da Esteira
   RUNG wire#powerrail
      Coil( "DauEes".EES001.LigEst )
   END_RUNG
   // the same network as SCL:
   "DauEes".EES001.LigEst := TRUE;
END_REGION

REGION Network 4: Definição da Peça
   RUNG wire#powerrail
      "DEFPEC"()
   END_RUNG
   // the same network as SCL:
   "DEFPEC"();
END_REGION

REGION Network 5: Seleção de peças do setor A
   RUNG wire#powerrail
      Contact( "DauEes".EES001_NewPec )
      { S7_Templates := "SrcType := Real" } EQ_Contact(in1 := "ParEes".EES001_PecMat, in2 := 1.0)
      wire#w1
      { S7_Templates := "SrcType := Real" } EQ_Contact(in1 := "ParEes".EES001_TamPec, in2 := 1.0)
      Contact( "DauEes".EES001_Sel.SetAPec01 )
      wire#w2
      Coil( "DauEes".EES001.AvnPiA )
   END_RUNG
   RUNG wire#w1
      { S7_Templates := "SrcType := Real" } EQ_Contact(in1 := "ParEes".EES001_TamPec, in2 := 2.0)
      Contact( "DauEes".EES001_Sel.SetAPec02 )
   END_RUNG wire#w2
   RUNG wire#w1
      { S7_Templates := "SrcType := Real" } EQ_Contact(in1 := "ParEes".EES001_TamPec, in2 := 3.0)
      Contact( "DauEes".EES001_Sel.SetAPec03 )
   END_RUNG wire#w2
   RUNG wire#powerrail
      Contact( "DauEes".EES001_NewPec )
      { S7_Templates := "SrcType := Real" } EQ_Contact(in1 := "ParEes".EES001_PecMat, in2 := 2.0)
      wire#w3
      { S7_Templates := "SrcType := Real" } EQ_Contact(in1 := "ParEes".EES001_TamPec, in2 := 1.0)
      Contact( "DauEes".EES001_Sel.SetAPec04 )
   END_RUNG wire#w2
   RUNG wire#w3
      { S7_Templates := "SrcType := Real" } EQ_Contact(in1 := "ParEes".EES001_TamPec, in2 := 2.0)
      Contact( "DauEes".EES001_Sel.SetAPec05 )
   END_RUNG wire#w2
   RUNG wire#w3
      { S7_Templates := "SrcType := Real" } EQ_Contact(in1 := "ParEes".EES001_TamPec, in2 := 3.0)
      Contact( "DauEes".EES001_Sel.SetAPec06 )
   END_RUNG wire#w2
   // the same network as SCL:
   "DauEes".EES001.AvnPiA := ("DauEes".EES001_NewPec AND ("ParEes".EES001_PecMat = 1.0) AND ((("ParEes".EES001_TamPec = 1.0) AND "DauEes".EES001_Sel.SetAPec01) OR (("ParEes".EES001_TamPec = 2.0) AND "DauEes".EES001_Sel.SetAPec02) OR (("ParEes".EES001_TamPec = 3.0) AND "DauEes".EES001_Sel.SetAPec03))) OR ("DauEes".EES001_NewPec AND ("ParEes".EES001_PecMat = 2.0) AND ((("ParEes".EES001_TamPec = 1.0) AND "DauEes".EES001_Sel.SetAPec04) OR (("ParEes".EES001_TamPec = 2.0) AND "DauEes".EES001_Sel.SetAPec05) OR (("ParEes".EES001_TamPec = 3.0) AND "DauEes".EES001_Sel.SetAPec06)));
END_REGION

REGION Network 6: Seleção de peças do setor B
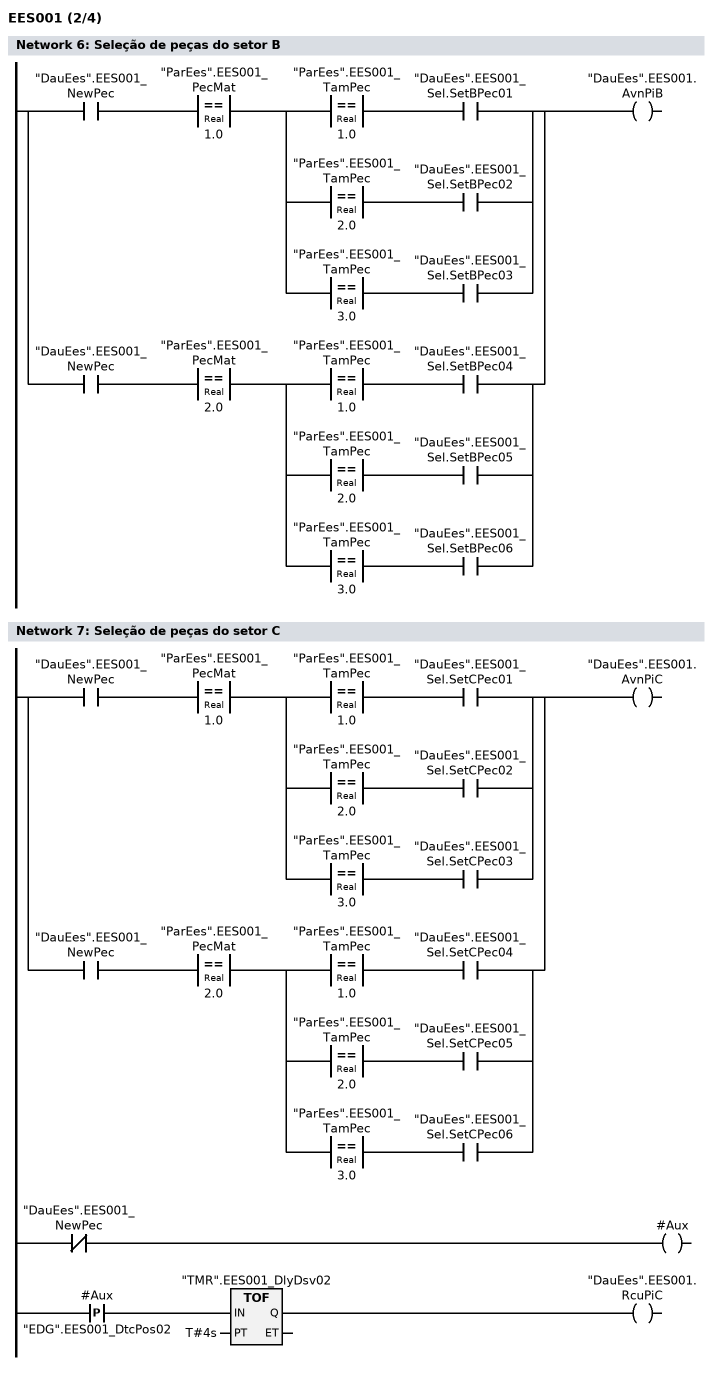
   RUNG wire#powerrail
      Contact( "DauEes".EES001_NewPec )
      { S7_Templates := "SrcType := Real" } EQ_Contact(in1 := "ParEes".EES001_PecMat, in2 := 1.0)
      wire#w1
      { S7_Templates := "SrcType := Real" } EQ_Contact(in1 := "ParEes".EES001_TamPec, in2 := 1.0)
      Contact( "DauEes".EES001_Sel.SetBPec01 )
      wire#w2
      Coil( "DauEes".EES001.AvnPiB )
   END_RUNG
   RUNG wire#w1
      { S7_Templates := "SrcType := Real" } EQ_Contact(in1 := "ParEes".EES001_TamPec, in2 := 2.0)
      Contact( "DauEes".EES001_Sel.SetBPec02 )
   END_RUNG wire#w2
   RUNG wire#w1
      { S7_Templates := "SrcType := Real" } EQ_Contact(in1 := "ParEes".EES001_TamPec, in2 := 3.0)
      Contact( "DauEes".EES001_Sel.SetBPec03 )
   END_RUNG wire#w2
   RUNG wire#powerrail
      Contact( "DauEes".EES001_NewPec )
      { S7_Templates := "SrcType := Real" } EQ_Contact(in1 := "ParEes".EES001_PecMat, in2 := 2.0)
      wire#w3
      { S7_Templates := "SrcType := Real" } EQ_Contact(in1 := "ParEes".EES001_TamPec, in2 := 1.0)
      Contact( "DauEes".EES001_Sel.SetBPec04 )
   END_RUNG wire#w2
   RUNG wire#w3
      { S7_Templates := "SrcType := Real" } EQ_Contact(in1 := "ParEes".EES001_TamPec, in2 := 2.0)
      Contact( "DauEes".EES001_Sel.SetBPec05 )
   END_RUNG wire#w2
   RUNG wire#w3
      { S7_Templates := "SrcType := Real" } EQ_Contact(in1 := "ParEes".EES001_TamPec, in2 := 3.0)
      Contact( "DauEes".EES001_Sel.SetBPec06 )
   END_RUNG wire#w2
   // the same network as SCL:
   "DauEes".EES001.AvnPiB := ("DauEes".EES001_NewPec AND ("ParEes".EES001_PecMat = 1.0) AND ((("ParEes".EES001_TamPec = 1.0) AND "DauEes".EES001_Sel.SetBPec01) OR (("ParEes".EES001_TamPec = 2.0) AND "DauEes".EES001_Sel.SetBPec02) OR (("ParEes".EES001_TamPec = 3.0) AND "DauEes".EES001_Sel.SetBPec03))) OR ("DauEes".EES001_NewPec AND ("ParEes".EES001_PecMat = 2.0) AND ((("ParEes".EES001_TamPec = 1.0) AND "DauEes".EES001_Sel.SetBPec04) OR (("ParEes".EES001_TamPec = 2.0) AND "DauEes".EES001_Sel.SetBPec05) OR (("ParEes".EES001_TamPec = 3.0) AND "DauEes".EES001_Sel.SetBPec06)));
END_REGION

REGION Network 7: Seleção de peças do setor C
   "DauEes".EES001.AvnPiC := ("DauEes".EES001_NewPec AND ("ParEes".EES001_PecMat = 1.0) AND ((("ParEes".EES001_TamPec = 1.0) AND "DauEes".EES001_Sel.SetCPec01) OR (("ParEes".EES001_TamPec = 2.0) AND "DauEes".EES001_Sel.SetCPec02) OR (("ParEes".EES001_TamPec = 3.0) AND "DauEes".EES001_Sel.SetCPec03))) OR ("DauEes".EES001_NewPec AND ("ParEes".EES001_PecMat = 2.0) AND ((("ParEes".EES001_TamPec = 1.0) AND "DauEes".EES001_Sel.SetCPec04) OR (("ParEes".EES001_TamPec = 2.0) AND "DauEes".EES001_Sel.SetCPec05) OR (("ParEes".EES001_TamPec = 3.0) AND "DauEes".EES001_Sel.SetCPec06)));
   #Aux := NOT "DauEes".EES001_NewPec;
   #_w1 := #Aux AND NOT "EDG".EES001_DtcPos02;   // rising edge of #Aux
   "EDG".EES001_DtcPos02 := #Aux;
   "TMR".EES001_DlyDsv02.TOF(IN := #_w1, PT := T#4s);
   "DauEes".EES001.RcuPiC := "TMR".EES001_DlyDsv02.Q;
END_REGION

REGION Network 8: Contador de peças do Setor A
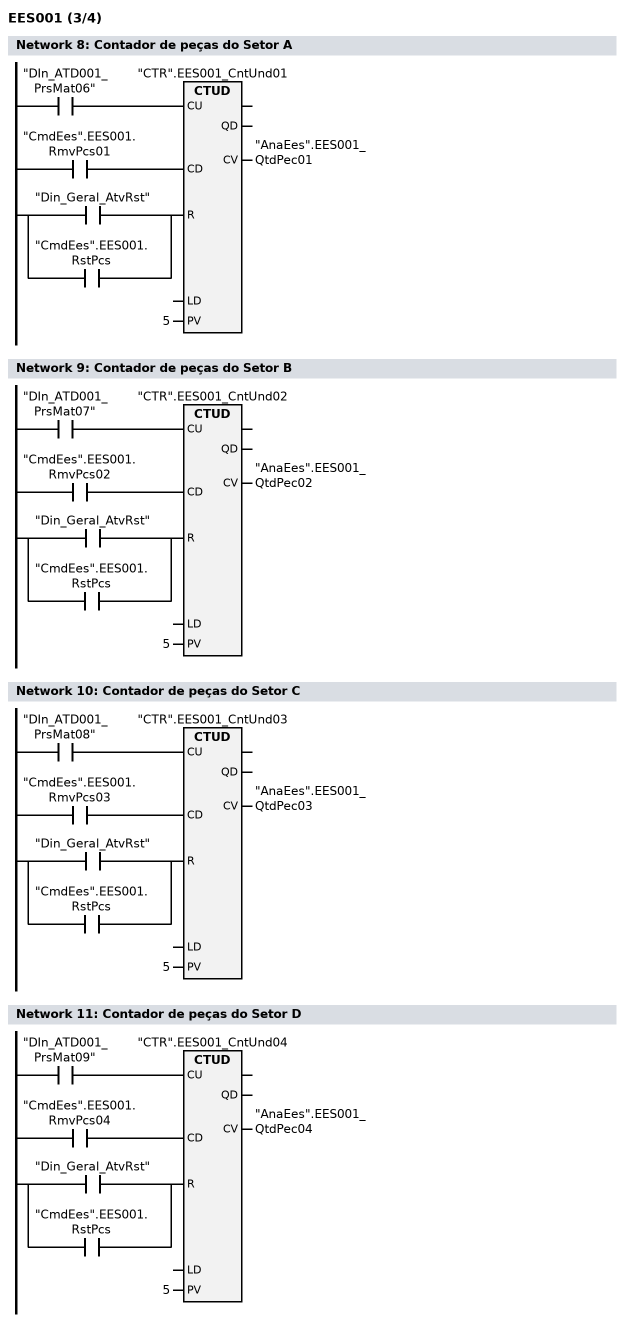
   "CTR".EES001_CntUnd01.CTUD(CU := "DIn_ATD001_PrsMat06",
                           CD := "CmdEes".EES001.RmvPcs01,
                           R := "Din_Geral_AtvRst" OR "CmdEes".EES001.RstPcs,
                           PV := 5,
                           CV => "AnaEes".EES001_QtdPec01);
END_REGION

REGION Network 9: Contador de peças do Setor B
   "CTR".EES001_CntUnd02.CTUD(CU := "DIn_ATD001_PrsMat07",
                           CD := "CmdEes".EES001.RmvPcs02,
                           R := "Din_Geral_AtvRst" OR "CmdEes".EES001.RstPcs,
                           PV := 5,
                           CV => "AnaEes".EES001_QtdPec02);
END_REGION

REGION Network 10: Contador de peças do Setor C
   "CTR".EES001_CntUnd03.CTUD(CU := "DIn_ATD001_PrsMat08",
                           CD := "CmdEes".EES001.RmvPcs03,
                           R := "Din_Geral_AtvRst" OR "CmdEes".EES001.RstPcs,
                           PV := 5,
                           CV => "AnaEes".EES001_QtdPec03);
END_REGION

REGION Network 11: Contador de peças do Setor D
   "CTR".EES001_CntUnd04.CTUD(CU := "DIn_ATD001_PrsMat09",
                           CD := "CmdEes".EES001.RmvPcs04,
                           R := "Din_Geral_AtvRst" OR "CmdEes".EES001.RstPcs,
                           PV := 5,
                           CV => "AnaEes".EES001_QtdPec04);
END_REGION

REGION Network 12: Calculo de Tempo de Transporte
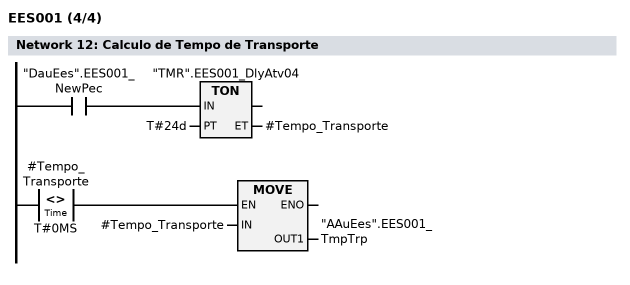
   "TMR".EES001_DlyAtv04.TON(IN := "DauEes".EES001_NewPec, PT := T#24d, ET => #Tempo_Transporte);
   IF #Tempo_Transporte <> T#0MS THEN "AAuEes".EES001_TmpTrp := #Tempo_Transporte; END_IF;
END_REGION
END_FUNCTION

// ===== PLC "PLCSim Adavanced"  CPU 1511-1 PN =====

VAR_GLOBAL   // PLC tag table "Default tag table"
   "Clock_Byte" AT %MB0 : Byte;
   "Clock_10Hz" AT %M0.0 : Bool;
   "Clock_5Hz" AT %M0.1 : Bool;
   "Clock_2.5Hz" AT %M0.2 : Bool;
   "Clock_2Hz" AT %M0.3 : Bool;
   "Clock_1.25Hz" AT %M0.4 : Bool;
   "Clock_1Hz" AT %M0.5 : Bool;
   "Clock_0.625Hz" AT %M0.6 : Bool;
   "Clock_0.5Hz" AT %M0.7 : Bool;
END_VAR

VAR_GLOBAL   // PLC tag table "Saídas Analógicas"
   "Dou_ATD001_LigElm01" AT %QD64 : Real;   // Esteira transportadora (ET-111) - Liga elemento (Esteira A)
   "Dou_ATD001_LigElm02" AT %QD68 : Real;   // Esteira transportadora (ET-111) - Liga elemento (Esteira B)
END_VAR

VAR_GLOBAL   // PLC tag table "Entradas Digitais"
   "DIn_ATD001_PrsMat01" AT %I20.0 : Bool;   // Esteira transportadora (ET-111) - Presença de material (tamanho maior)
   "DIn_ATD001_PrsMat02" AT %I20.1 : Bool;   // Esteira transportadora (ET-111) - Presença de material (tamanho médio)
   "DIn_ATD001_PrsMat03" AT %I20.2 : Bool;   // Esteira transportadora (ET-111) - Presença de material (tamanho menor)
   "DIn_ATD001_PrsMat04" AT %I20.3 : Bool;   // Esteira transportadora (ET-111) - Presença de material (Capacitivo)
   "DIn_ATD001_PrsMat05" AT %I20.4 : Bool;   // Esteira transportadora (ET-111) - Presença de material (Indutivo)
   "DIn_ATD001_PrsMat06" AT %I20.5 : Bool;   // Esteira transportadora (ET-111) - Presença de material (Setor A)
   "DIn_ATD001_PrsMat07" AT %I20.6 : Bool;   // Esteira transportadora (ET-111) - Presença de material (Setor B)
   "DIn_ATD001_PrsMat08" AT %I20.7 : Bool;   // Esteira transportadora (ET-111) - Presença de material (Setor C)
   "DIn_ATD001_PrsMat09" AT %I21.0 : Bool;   // Esteira transportadora (ET-111) - Presença de material (Setor D)
   "Din_Geral_AtvEmg" AT %I21.1 : Bool;   // Geral - Ativa condição de emergência [NF]
   "Din_Geral_AtvRst" AT %I21.2 : Bool;   // Geral - Ativa reset
END_VAR

VAR_GLOBAL   // PLC tag table "Saídas Digitais"
   "Dou_ATD002_AvnElm" AT %Q20.0 : Bool;   // Pistão Separador A (PI-111) - Avança elemento
   "Dou_ATD003_AvnElm" AT %Q20.1 : Bool;   // Pistão Separador B (PI-112) - Avança elemento
   "Dou_ATD004_AvnElm" AT %Q20.2 : Bool;   // Pistão Separador C (PI-113) - Avança elemento
   "Dou_ATD004_RcuElm" AT %Q20.3 : Bool;   // Pistão Separador C (PI-113) - Recua elemento
END_VAR

// folder: System blocks/Program resources

DATA_BLOCK "EES001_DlyDsv01"   // DB4
{ S7_Optimized_Access := 'TRUE' }
AUTHOR : Simatic
FAMILY : IEC
NAME : IEC_TMR
VERSION : 1.0
// stored: InstanceOfName IEC_TIMER
"IEC_TIMER"
BEGIN
END_DATA_BLOCK

// folder: VARIÁVEIS/0 - Gerais

DATA_BLOCK "EDG"   // DB1
TITLE = Detecção de Bordas
{ S7_Optimized_Access := 'TRUE' }
VERSION : 0.1
   VAR
      GRP001_DtcPos01 : Bool;   // Geral - Detecção positiva
      EES001_DtcPos01 : Bool;   // Selecionador de Peças - Detecção positiva
      EES001_DtcPos02 : Bool;   // Selecionador de Peças - Detecção positiva (Aux)
      EES001_DtcPos03 : Bool;   // Selecionador de Peças - Detecção positiva (Tempo de transporte)
   END_VAR
BEGIN
END_DATA_BLOCK

DATA_BLOCK "TMR"   // DB2
TITLE = Temporizadores
{ S7_Optimized_Access := 'TRUE' }
VERSION : 0.1
   VAR
      EES001_DlyAtv01 : IEC_TIMER;   // Selecionador de Peças - Atraso para ativar
      EES001_DlyAtv02 : IEC_TIMER;   // Selecionador de Peças - Atraso para ativar
      EES001_DlyAtv03 : IEC_TIMER;   // Selecionador de Peças - Atraso para ativar
      ATD003_DlyAtv01 : IEC_TIMER;   // Pistão Separador B - Atraso para ativar
      EES001_DlyDsv01 : IEC_TIMER;   // Selecionador de Peças - Atraso para desativar
      EES001_DlyDsv02 : IEC_TIMER;   // Selecionador de Peças - Atraso para desativar (Recuar Pistão C)
      ATD004_DlyAtv01 : IEC_TIMER;   // Pistão Separador C - Atraso para ativar (Avançar)
      EES001_DlyAtv04 : IEC_TIMER;   // Selecionador de Peças - Atraso para ativar (Tempo de transporte)
   END_VAR
BEGIN
END_DATA_BLOCK

DATA_BLOCK "CTR"   // DB3
TITLE = Contadores
{ S7_Optimized_Access := 'TRUE' }
VERSION : 0.1
   VAR
      EES001_CntUnd01 : IEC_UCOUNTER;   // Selecionador de Peças - Conta unidades (Setor A)
      EES001_CntUnd02 : IEC_UCOUNTER;   // Selecionador de Peças - Conta unidades (Setor B)
      EES001_CntUnd03 : IEC_UCOUNTER;   // Selecionador de Peças - Conta unidades (Setor C)
      EES001_CntUnd04 : IEC_UCOUNTER;   // Selecionador de Peças - Conta unidades (Setor D)
   END_VAR
BEGIN
END_DATA_BLOCK

// folder: VARIÁVEIS/1 - Comandos

DATA_BLOCK "CmdEsp"   // DB110
{ S7_Optimized_Access := 'FALSE' }
VERSION : 0.1
BEGIN
END_DATA_BLOCK

DATA_BLOCK "CmdGrp"   // DB120
{ S7_Optimized_Access := 'FALSE' }
VERSION : 0.1
   VAR
      GRP001 : Struct   // Geral
         RrmElm : Bool := false;   // Geral - Rearma Elemento
         SelAut : Bool := false;   // Geral - Seleciona modo automático para todos atuadores
         SelMaa : Bool := false;   // Geral - Seleciona modo manual para todos atuadores
         xd0r3 : Bool := false;   // Reserva
         xd0r4 : Bool := false;   // Reserva
         xd0r5 : Bool := false;   // Reserva
         xd0r6 : Bool := false;   // Reserva
         xd0r7 : Bool := false;   // Reserva
         xd1r0 : Bool := false;   // Reserva
         xd1r1 : Bool := false;   // Reserva
         xd1r2 : Bool := false;   // Reserva
         xd1r3 : Bool := false;   // Reserva
         xd1r4 : Bool := false;   // Reserva
         xd1r5 : Bool := false;   // Reserva
         xd1r6 : Bool := false;   // Reserva
         xd1r7 : Bool := false;   // Reserva
      END_STRUCT;
   END_VAR
BEGIN
END_DATA_BLOCK

DATA_BLOCK "CmdAtd"   // DB130
TITLE = Comandos
{ S7_Optimized_Access := 'FALSE' }
VERSION : 0.1
   VAR
      ATD001 : Struct   // Esteira Transportadora (ET-111)
         SelAut : Bool;   // Esteira Transportadora (ET-111) - Seleciona modo automático
         SelMaa : Bool := false;   // Esteira Transportadora (ET-111) - Seleciona modo manual
         LigElm : Bool := false;   // Esteira Transportadora (ET-111) - Liga elemento
         DsgElm : Bool := false;   // Esteira Transportadora (ET-111) - Desliga elemento
         xd0r4 : Bool := false;   // Reserva
         xd0r5 : Bool := false;   // Reserva
         xd0r6 : Bool := false;   // Reserva
         xd0r7 : Bool := false;   // Reserva
         xd1r0 : Bool;   // Reserva
         xd1r1 : Bool := false;   // Reserva
         xd1r2 : Bool := false;   // Reserva
         xd1r3 : Bool := false;   // Reserva
         xd1r4 : Bool := false;   // Reserva
         xd1r5 : Bool := false;   // Reserva
         xd1r6 : Bool := false;   // Reserva
         xd1r7 : Bool := false;   // Reserva
      END_STRUCT;
      ATD002 : Struct   // Pistão Separador A (PI-111)
         SelAut : Bool := false;   // Pistão Separador A (PI-111) - Seleciona modo automático
         SelMaa : Bool := false;   // Pistão Separador A (PI-111) - Seleciona modo manual
         AvnElm : Bool := false;   // Pistão Separador A (PI-111) - Avança elemento
         RcuElm : Bool := false;   // Pistão Separador A (PI-111) - Recua elemento
         xd0r4 : Bool := false;   // Reserva
         xd0r5 : Bool := false;   // Reserva
         xd0r6 : Bool := false;   // Reserva
         xd0r7 : Bool := false;   // Reserva
         xd1r0 : Bool := false;   // Reserva
         xd1r1 : Bool := false;   // Reserva
         xd1r2 : Bool := false;   // Reserva
         xd1r3 : Bool := false;   // Reserva
         xd1r4 : Bool := false;   // Reserva
         xd1r5 : Bool := false;   // Reserva
         xd1r6 : Bool := false;   // Reserva
         xd1r7 : Bool := false;   // Reserva
      END_STRUCT;
      ATD003 : Struct   // Pistão Separador B (PI-112)
         SelAut : Bool := false;   // Pistão Separador B (PI-112) - Seleciona modo automático
         SelMaa : Bool := false;   // Pistão Separador B (PI-112) - Seleciona modo manual
         AvnElm : Bool := false;   // Pistão Separador B (PI-112) - Avança elemento
         RcuElm : Bool := false;   // Pistão Separador B (PI-112) - Recua elemento
         xd0r4 : Bool := false;   // Reserva
         xd0r5 : Bool := false;   // Reserva
         xd0r6 : Bool := false;   // Reserva
         xd0r7 : Bool := false;   // Reserva
         xd1r0 : Bool := false;   // Reserva
         xd1r1 : Bool := false;   // Reserva
         xd1r2 : Bool := false;   // Reserva
         xd1r3 : Bool := false;   // Reserva
         xd1r4 : Bool := false;   // Reserva
         xd1r5 : Bool := false;   // Reserva
         xd1r6 : Bool := false;   // Reserva
         xd1r7 : Bool := false;   // Reserva
      END_STRUCT;
      ATD004 : Struct   // Pistão Separador C (PI-113)
         SelAut : Bool := false;   // Pistão Separador C (PI-113) - Seleciona modo automático
         SelMaa : Bool := false;   // Pistão Separador C (PI-113) - Seleciona modo manual
         AvnElm : Bool := false;   // Pistão Separador C (PI-113) - Avança elemento
         RcuElm : Bool := false;   // Pistão Separador C (PI-113) - Recua elemento
         xd0r4 : Bool := false;   // Reserva
         xd0r5 : Bool := false;   // Reserva
         xd0r6 : Bool := false;   // Reserva
         xd0r7 : Bool := false;   // Reserva
         xd1r0 : Bool := false;   // Reserva
         xd1r1 : Bool := false;   // Reserva
         xd1r2 : Bool := false;   // Reserva
         xd1r3 : Bool := false;   // Reserva
         xd1r4 : Bool := false;   // Reserva
         xd1r5 : Bool := false;   // Reserva
         xd1r6 : Bool := false;   // Reserva
         xd1r7 : Bool := false;   // Reserva
      END_STRUCT;
   END_VAR
BEGIN
END_DATA_BLOCK

DATA_BLOCK "CmdEes"   // DB160
{ S7_Optimized_Access := 'FALSE' }
VERSION : 0.1
   VAR
      EES001 : Struct   // Selecionador de Peças
         RrmElm : Bool := false;   // Selecionador de Peças - Rearma Elmento
         RmvPcs01 : Bool := false;   // Selecionador de Peças - Remove Peças (Setor A)
         RmvPcs02 : Bool := false;   // Selecionador de Peças - Remove Peças (Setor B)
         RmvPcs03 : Bool := false;   // Selecionador de Peças - Remove Peças (Setor C)
         RmvPcs04 : Bool := false;   // Selecionador de Peças - Remove Peças (Setor D)
         RstPcs : Bool := false;   // Selecionador de Peças - Reseta quantidade de Peças
         xd0r6 : Bool := false;   // Reserva
         xd0r7 : Bool := false;   // Reserva
         xd1r0 : Bool := false;   // Reserva
         xd1r1 : Bool := false;   // Reserva
         xd1r2 : Bool := false;   // Reserva
         xd1r3 : Bool := false;   // Reserva
         xd1r4 : Bool := false;   // Reserva
         xd1r5 : Bool := false;   // Reserva
         xd1r6 : Bool := false;   // Reserva
         xd1r7 : Bool := false;   // Reserva
      END_STRUCT;
   END_VAR
BEGIN
END_DATA_BLOCK

// folder: VARIÁVEIS/2 - Estados

DATA_BLOCK "SttEsp"   // DB210
{ S7_Optimized_Access := 'FALSE' }
VERSION : 0.1
BEGIN
END_DATA_BLOCK

DATA_BLOCK "SttGrp"   // DB220
{ S7_Optimized_Access := 'FALSE' }
VERSION : 0.1
   VAR
      GRP001 : Struct   // Geral
         xd0r0 : Bool := false;   // Reserva
         xd0r1 : Bool := false;   // Reserva
         xd0r2 : Bool := false;   // Reserva
         xd0r3 : Bool := false;   // Reserva
         xd0r4 : Bool := false;   // Reserva
         xd0r5 : Bool := false;   // Reserva
         xd0r6 : Bool := false;   // Reserva
         xd0r7 : Bool := false;   // Reserva
         xd1r0 : Bool := false;   // Reserva
         xd1r1 : Bool := false;   // Reserva
         xd1r2 : Bool := false;   // Reserva
         xd1r3 : Bool := false;   // Reserva
         xd1r4 : Bool := false;   // Reserva
         xd1r5 : Bool := false;   // Reserva
         xd1r6 : Bool := false;   // Reserva
         xd1r7 : Bool := false;   // Reserva
      END_STRUCT;
   END_VAR
BEGIN
END_DATA_BLOCK

DATA_BLOCK "SttAtd"   // DB230
TITLE = Estados de Atuadores
{ S7_Optimized_Access := 'FALSE' }
VERSION : 0.1
   VAR
      ATD001 : Struct   // Esteira Transportadora (ET-111)
         AutSel : Bool := false;   // Esteira Transportadora (ET-111) - Modo automático selecionado
         MaaSel : Bool := false;   // Esteira Transportadora (ET-111) - Modo manual selecionado
         ElmLig : Bool := false;   // Esteira Transportadora (ET-111) - Elemento ligado
         BlqLig : Bool := false;   // Esteira Transportadora (ET-111) - Bloqueado para ligar
         xd0r4 : Bool := false;   // Reserva
         xd0r5 : Bool := false;   // Reserva
         xd0r6 : Bool := false;   // Reserva
         xd0r7 : Bool := false;   // Reserva
         xd1r0 : Bool := false;   // Reserva
         xd1r1 : Bool := false;   // Reserva
         xd1r2 : Bool := false;   // Reserva
         xd1r3 : Bool := false;   // Reserva
         xd1r4 : Bool := false;   // Reserva
         xd1r5 : Bool := false;   // Reserva
         xd1r6 : Bool := false;   // Reserva
         xd1r7 : Bool := false;   // Reserva
      END_STRUCT;
      ATD002 : Struct   // Pistão Separador A (PI-111)
         AutSel : Bool := false;   // Pistão Separador A (PI-111) - Modo automático selecionado
         MaaSel : Bool := false;   // Pistão Separador A (PI-111) - Modo manual selecionado
         PosAvn : Bool := false;   // Pistão Separador A (PI-111) - Elemento avançado
         BlqAvn : Bool := false;   // Pistão Separador A (PI-111) - Bloqueado para avançar
         xd0r4 : Bool := false;   // Reserva
         xd0r5 : Bool := false;   // Reserva
         xd0r6 : Bool := false;   // Reserva
         xd0r7 : Bool := false;   // Reserva
         xd1r0 : Bool := false;   // Reserva
         xd1r1 : Bool := false;   // Reserva
         xd1r2 : Bool := false;   // Reserva
         xd1r3 : Bool := false;   // Reserva
         xd1r4 : Bool := false;   // Reserva
         xd1r5 : Bool := false;   // Reserva
         xd1r6 : Bool := false;   // Reserva
         xd1r7 : Bool := false;   // Reserva
      END_STRUCT;
      ATD003 : Struct   // Pistão Separador B (PI-112)
         AutSel : Bool := false;   // Pistão Separador B (PI-112) - Modo automático selecionado
         MaaSel : Bool := false;   // Pistão Separador B (PI-112) - Modo manual selecionado
         PosAvn : Bool := false;   // Pistão Separador B (PI-112) - Elemento avançado
         BlqAvn : Bool := false;   // Pistão Separador B (PI-112) - Bloqueado para Bloqueado para avançar
         xd0r4 : Bool := false;   // Reserva
         xd0r5 : Bool := false;   // Reserva
         xd0r6 : Bool := false;   // Reserva
         xd0r7 : Bool := false;   // Reserva
         xd1r0 : Bool := false;   // Reserva
         xd1r1 : Bool := false;   // Reserva
         xd1r2 : Bool := false;   // Reserva
         xd1r3 : Bool := false;   // Reserva
         xd1r4 : Bool := false;   // Reserva
         xd1r5 : Bool := false;   // Reserva
         xd1r6 : Bool := false;   // Reserva
         xd1r7 : Bool := false;   // Reserva
      END_STRUCT;
      ATD004 : Struct   // Pistão Separador C (PI-113)
         AutSel : Bool := false;   // Pistão Separador C (PI-113) - Modo automático selecionado
         MaaSel : Bool := false;   // Pistão Separador C (PI-113) - Modo manual selecionado
         PosAvn : Bool := false;   // Pistão Separador C (PI-113) - Elemento avançado
         BlqAvn : Bool := false;   // Pistão Separador C (PI-113) - Bloqueado para avançar
         PosRcu : Bool := false;   // Pistão Separador C (PI-113) - Elemento recuado
         BlqRcu : Bool := false;   // Pistão Separador C (PI-113) - Bloqueado para recuar
         xd0r6 : Bool := false;   // Reserva
         xd0r7 : Bool := false;   // Reserva
         xd1r0 : Bool := false;   // Reserva
         xd1r1 : Bool := false;   // Reserva
         xd1r2 : Bool := false;   // Reserva
         xd1r3 : Bool := false;   // Reserva
         xd1r4 : Bool := false;   // Reserva
         xd1r5 : Bool := false;   // Reserva
         xd1r6 : Bool := false;   // Reserva
         xd1r7 : Bool := false;   // Reserva
      END_STRUCT;
   END_VAR
BEGIN
END_DATA_BLOCK

DATA_BLOCK "SttEes"   // DB260
{ S7_Optimized_Access := 'FALSE' }
VERSION : 0.1
   VAR
      EES001 : Struct   // Selecionador de Peças
         ElmDef : Bool := false;   // Selecionador de Peças - Elmento com Defeito
         xd0r1 : Bool := false;   // Reserva
         xd0r2 : Bool := false;   // Reserva
         xd0r3 : Bool := false;   // Reserva
         xd0r4 : Bool := false;   // Reserva
         xd0r5 : Bool := false;   // Reserva
         xd0r6 : Bool := false;   // Reserva
         xd0r7 : Bool := false;   // Reserva
         xd1r0 : Bool := false;   // Reserva
         xd1r1 : Bool := false;   // Reserva
         xd1r2 : Bool := false;   // Reserva
         xd1r3 : Bool := false;   // Reserva
         xd1r4 : Bool := false;   // Reserva
         xd1r5 : Bool := false;   // Reserva
         xd1r6 : Bool := false;   // Reserva
         xd1r7 : Bool := false;   // Reserva
      END_STRUCT;
   END_VAR
BEGIN
END_DATA_BLOCK

// folder: VARIÁVEIS/3 - Alarmes

DATA_BLOCK "AlrEsp"   // DB310
{ S7_Optimized_Access := 'FALSE' }
VERSION : 0.1
BEGIN
END_DATA_BLOCK

DATA_BLOCK "AlrGrp"   // DB320
{ S7_Optimized_Access := 'FALSE' }
VERSION : 0.1
   VAR
      GRP001 : Struct   // Geral
         EmgAtv : Bool := false;   // Geral - Condição de Emergência Ativada
         xd0r1 : Bool := false;   // Reserva
         xd0r2 : Bool := false;   // Reserva
         xd0r3 : Bool := false;   // Reserva
         xd0r4 : Bool := false;   // Reserva
         xd0r5 : Bool := false;   // Reserva
         xd0r6 : Bool := false;   // Reserva
         xd0r7 : Bool := false;   // Reserva
         xd1r0 : Bool := false;   // Reserva
         xd1r1 : Bool := false;   // Reserva
         xd1r2 : Bool := false;   // Reserva
         xd1r3 : Bool := false;   // Reserva
         xd1r4 : Bool := false;   // Reserva
         xd1r5 : Bool := false;   // Reserva
         xd1r6 : Bool := false;   // Reserva
         xd1r7 : Bool := false;   // Reserva
      END_STRUCT;
   END_VAR
BEGIN
END_DATA_BLOCK

DATA_BLOCK "AlrAtd"   // DB330
TITLE = Alarmes de Atuadores
{ S7_Optimized_Access := 'FALSE' }
VERSION : 0.1
   VAR
      ATD001 : Struct   // Esteira Transportadora (ET-111)
         xd0r0 : Bool := false;   // Reserva
         xd0r1 : Bool := false;   // Reserva
         xd0r2 : Bool := false;   // Reserva
         xd0r3 : Bool := false;   // Reserva
         xd0r4 : Bool := false;   // Reserva
         xd0r5 : Bool := false;   // Reserva
         xd0r6 : Bool := false;   // Reserva
         xd0r7 : Bool := false;   // Reserva
         xd1r0 : Bool := false;   // Reserva
         xd1r1 : Bool := false;   // Reserva
         xd1r2 : Bool := false;   // Reserva
         xd1r3 : Bool := false;   // Reserva
         xd1r4 : Bool := false;   // Reserva
         xd1r5 : Bool := false;   // Reserva
         xd1r6 : Bool := false;   // Reserva
         xd1r7 : Bool := false;   // Reserva
      END_STRUCT;
      ATD002 : Struct   // Pistão Separador A (PI-111)
         xd0r0 : Bool := false;   // Reserva
         xd0r1 : Bool := false;   // Reserva
         xd0r2 : Bool := false;   // Reserva
         xd0r3 : Bool := false;   // Reserva
         xd0r4 : Bool := false;   // Reserva
         xd0r5 : Bool := false;   // Reserva
         xd0r6 : Bool := false;   // Reserva
         xd0r7 : Bool := false;   // Reserva
         xd1r0 : Bool := false;   // Reserva
         xd1r1 : Bool := false;   // Reserva
         xd1r2 : Bool := false;   // Reserva
         xd1r3 : Bool := false;   // Reserva
         xd1r4 : Bool := false;   // Reserva
         xd1r5 : Bool := false;   // Reserva
         xd1r6 : Bool := false;   // Reserva
         xd1r7 : Bool := false;   // Reserva
      END_STRUCT;
      ATD003 : Struct   // Pistão Separador B (PI-112)
         xd0r0 : Bool := false;   // Reserva
         xd0r1 : Bool := false;   // Reserva
         xd0r2 : Bool := false;   // Reserva
         xd0r3 : Bool := false;   // Reserva
         xd0r4 : Bool := false;   // Reserva
         xd0r5 : Bool := false;   // Reserva
         xd0r6 : Bool := false;   // Reserva
         xd0r7 : Bool := false;   // Reserva
         xd1r0 : Bool := false;   // Reserva
         xd1r1 : Bool := false;   // Reserva
         xd1r2 : Bool := false;   // Reserva
         xd1r3 : Bool := false;   // Reserva
         xd1r4 : Bool := false;   // Reserva
         xd1r5 : Bool := false;   // Reserva
         xd1r6 : Bool := false;   // Reserva
         xd1r7 : Bool := false;   // Reserva
      END_STRUCT;
      ATD004 : Struct   // Pistão Separador C (PI-113)
         xd0r0 : Bool := false;   // Reserva
         xd0r1 : Bool := false;   // Reserva
         xd0r2 : Bool := false;   // Reserva
         xd0r3 : Bool := false;   // Reserva
         xd0r4 : Bool := false;   // Reserva
         xd0r5 : Bool := false;   // Reserva
         xd0r6 : Bool := false;   // Reserva
         xd0r7 : Bool := false;   // Reserva
         xd1r0 : Bool := false;   // Reserva
         xd1r1 : Bool := false;   // Reserva
         xd1r2 : Bool := false;   // Reserva
         xd1r3 : Bool := false;   // Reserva
         xd1r4 : Bool := false;   // Reserva
         xd1r5 : Bool := false;   // Reserva
         xd1r6 : Bool := false;   // Reserva
         xd1r7 : Bool := false;   // Reserva
      END_STRUCT;
   END_VAR
BEGIN
END_DATA_BLOCK

